KUKA KRL program: MyProgram_120().src

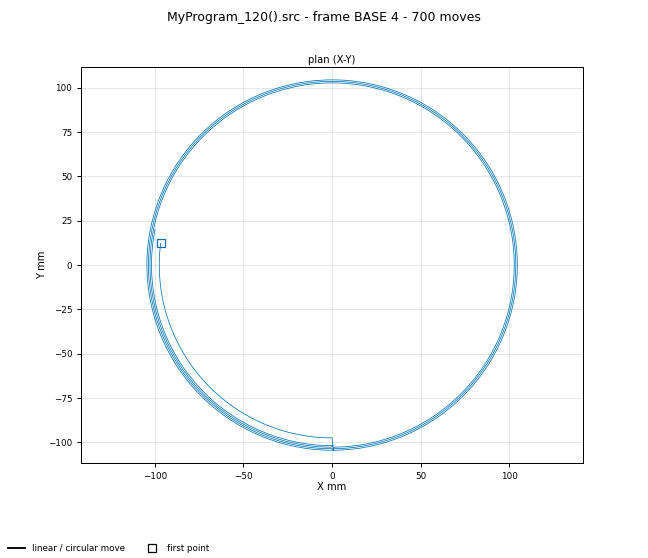
[picture p0: tool path of MyProgram_120().src in frame BASE 4, 700 of 700 moves have a stored position in this frame; points joined in program order, loops and branches not executed]
&ACCESS RVP
&REL 1
&PARAM TEMPLATE = C:\KRC\Roboter\Template\vorgabe
&PARAM EDITMASK = *
DEF MyProgram_120()
; ---- Setting reference (Base) ----
$BASE = BASE_DATA[4]

; --------------------------
; ---- Setting tool (TCP) ----
$TOOL = TOOL_DATA[3]
; --------------------------

$VEL.CP = VEL_APROX_PRINT
Startdeposition()
$VEL.CP = VEL_PRINT
LIN {X -96.7229,Y 12.2113,Z 101,A 168.4745,B 24.9259,C -1.9878,E1 24.8409,E2 276.8389} C_DIS
LIN {X -97.0219,Y 9.5617,Z 101,A 170.028,B 24.9263,C -1.9823,E1 24.8405,E2 275.2892} C_DIS
LIN {X -97.2007,Y 7.5113,Z 101,A 171.291,B 24.9265,C -1.9802,E1 24.8402,E2 274.0237} C_DIS
LIN {X -97.3722,Y 4.8262,Z 101,A 172.8402,B 24.9269,C -1.974,E1 24.8399,E2 272.4798} C_DIS
LIN {X -97.4611,Y 2.4408,Z 101,A 174.2525,B 24.9272,C -1.9698,E1 24.8399,E2 271.0691} C_DIS
LIN {X -97.4919,Y 0.0083,Z 101,A 175.6921,B 24.9276,C -1.9656,E1 24.8398,E2 269.631} C_DIS
LIN {X -97.4637,Y -2.3325,Z 101,A 177.0782,B 24.9279,C -1.9615,E1 24.8398,E2 268.2463} C_DIS
LIN {X -97.3763,Y -4.7434,Z 101,A 178.5071,B 24.9282,C -1.9573,E1 24.84,E2 266.8188} C_DIS
LIN {X -97.231,Y -7.125,Z 101,A 179.9181,B 24.9285,C -1.9531,E1 24.8403,E2 265.4093} C_DIS
LIN {X -97.0288,Y -9.488,Z 101,A -178.679,B 24.9288,C -1.949,E1 24.8407,E2 264.0078} C_DIS
LIN {X -96.7605,Y -11.9197,Z 101,A -177.2313,B 24.9291,C -1.9447,E1 24.8411,E2 262.5616} C_DIS
LIN {X -96.4472,Y -14.2312,Z 101,A -175.8498,B 24.9294,C -1.9408,E1 24.8417,E2 261.1814} C_DIS
LIN {X -96.0565,Y -16.6684,Z 101,A -174.3908,B 24.9297,C -1.9365,E1 24.8423,E2 259.7239} C_DIS
LIN {X -95.6192,Y -19.017,Z 101,A -172.9768,B 24.93,C -1.9324,E1 24.8431,E2 258.3112} C_DIS
LIN {X -95.1138,Y -21.401,Z 101,A -171.3294,B 24.9298,C -1.9351,E1 24.8441,E2 256.6478} C_DIS
LIN {X -94.2834,Y -24.8046,Z 101,A -169.4616,B 24.9307,C -1.9225,E1 24.8453,E2 254.7992} C_DIS
LIN {X -93.6343,Y -27.1534,Z 101,A -168.0199,B 24.931,C -1.9184,E1 24.8464,E2 253.3587} C_DIS
LIN {X -92.6398,Y -30.37,Z 101,A -166.0424,B 24.9314,C -1.9125,E1 24.8481,E2 251.3841} C_DIS
LIN {X -91.9528,Y -32.3885,Z 101,A -164.6967,B 24.9314,C -1.9118,E1 24.8493,E2 250.0322} C_DIS
LIN {X -90.9778,Y -35.038,Z 101,A -163.097,B 24.932,C -1.905,E1 24.8509,E2 248.4399} C_DIS
LIN {X -90.0939,Y -37.2519,Z 101,A -161.6859,B 24.9322,C -1.9012,E1 24.8524,E2 247.0298} C_DIS
LIN {X -89.1565,Y -39.4427,Z 101,A -160.2806,B 24.9325,C -1.8974,E1 24.854,E2 245.626} C_DIS
LIN {X -88.1312,Y -41.6842,Z 101,A -158.8206,B 24.9328,C -1.8937,E1 24.8557,E2 244.1668} C_DIS
LIN {X -87.104,Y -43.7895,Z 101,A -157.4349,B 24.933,C -1.8902,E1 24.8574,E2 242.7821} C_DIS
LIN {X -86.005,Y -45.9104,Z 101,A -155.8779,B 24.933,C -1.8914,E1 24.8594,E2 241.2139} C_DIS
LIN {X -84.4429,Y -48.7212,Z 101,A -154.0565,B 24.9335,C -1.8841,E1 24.8619,E2 239.4005} C_DIS
LIN {X -82.9985,Y -51.1462,Z 101,A -152.4547,B 24.9339,C -1.8777,E1 24.8642,E2 237.8055} C_DIS
LIN {X -81.8862,Y -52.9061,Z 101,A -151.1887,B 24.934,C -1.876,E1 24.8662,E2 236.5372} C_DIS
LIN {X -79.7344,Y -56.0986,Z 101,A -148.9459,B 24.9345,C -1.8696,E1 24.8697,E2 234.2985} C_DIS
LIN {X -78.3085,Y -58.0728,Z 101,A -147.5081,B 24.9347,C -1.8663,E1 24.8721,E2 232.8617} C_DIS
LIN {X -76.7454,Y -60.1219,Z 101,A -145.8271,B 24.9346,C -1.8683,E1 24.875,E2 231.1679} C_DIS
LIN {X -74.5735,Y -62.7968,Z 101,A -143.7539,B 24.9348,C -1.8652,E1 24.8787,E2 229.0926} C_DIS
LIN {X -72.2811,Y -65.4221,Z 101,A -141.6893,B 24.9351,C -1.8611,E1 24.8825,E2 227.0285} C_DIS
LIN {X -70.1933,Y -67.6552,Z 101,A -139.9774,B 24.9355,C -1.8543,E1 24.8858,E2 225.3253} C_DIS
LIN {X -67.6749,Y -70.1743,Z 101,A -137.8668,B 24.9358,C -1.8505,E1 24.89,E2 223.2149} C_DIS
LIN {X -65.0221,Y -72.6391,Z 101,A -135.7428,B 24.9361,C -1.8461,E1 24.8943,E2 221.0927} C_DIS
LIN {X -62.3326,Y -74.9598,Z 101,A -133.6387,B 24.9364,C -1.8427,E1 24.8988,E2 218.9887} C_DIS
LIN {X -59.5972,Y -77.1525,Z 101,A -131.585,B 24.9366,C -1.8387,E1 24.9033,E2 216.9369} C_DIS
LIN {X -57.1512,Y -78.9834,Z 101,A -129.8771,B 24.9371,C -1.8326,E1 24.9071,E2 215.2376} C_DIS
LIN {X -55.1551,Y -80.3903,Z 101,A -128.4366,B 24.9372,C -1.8304,E1 24.9105,E2 213.7974} C_DIS
LIN {X -53.1374,Y -81.7378,Z 101,A -126.7931,B 24.9368,C -1.8357,E1 24.9143,E2 212.1358} C_DIS
LIN {X -50.1638,Y -83.5955,Z 101,A -124.9406,B 24.9375,C -1.8254,E1 24.9187,E2 210.3021} C_DIS
LIN {X -48.0882,Y -84.8066,Z 101,A -123.5216,B 24.9377,C -1.8236,E1 24.9221,E2 208.8832} C_DIS
LIN {X -45.9565,Y -85.9807,Z 101,A -122.0876,B 24.9377,C -1.8218,E1 24.9257,E2 207.4493} C_DIS
LIN {X -42.7678,Y -87.6104,Z 101,A -119.9768,B 24.938,C -1.8194,E1 24.9309,E2 205.3386} C_DIS
LIN {X -40.652,Y -88.6117,Z 101,A -118.5977,B 24.938,C -1.818,E1 24.9344,E2 203.9595} C_DIS
LIN {X -38.4283,Y -89.5987,Z 101,A -117.1645,B 24.9381,C -1.8166,E1 24.9381,E2 202.5263} C_DIS
LIN {X -36.5181,Y -90.3926,Z 101,A -115.9075,B 24.9381,C -1.8168,E1 24.9413,E2 201.2659} C_DIS
LIN {X -34.0204,Y -91.3632,Z 101,A -114.3685,B 24.9383,C -1.8141,E1 24.9453,E2 199.7302} C_DIS
LIN {X -31.8745,Y -92.1332,Z 101,A -113.0168,B 24.9383,C -1.8134,E1 24.9489,E2 198.3775} C_DIS
LIN {X -29.4455,Y -92.9389,Z 101,A -111.5188,B 24.9385,C -1.812,E1 24.9529,E2 196.8801} C_DIS
LIN {X -27.1599,Y -93.6323,Z 101,A -110.1131,B 24.9385,C -1.8111,E1 24.9567,E2 195.4743} C_DIS
LIN {X -24.8583,Y -94.2695,Z 101,A -108.7074,B 24.9385,C -1.8103,E1 24.9604,E2 194.0682} C_DIS
LIN {X -22.864,Y -94.7714,Z 101,A -107.4594,B 24.9385,C -1.811,E1 24.9638,E2 192.8167} C_DIS
LIN {X -20.1943,Y -95.3775,Z 101,A -105.8867,B 24.9387,C -1.809,E1 24.9681,E2 191.2469} C_DIS
LIN {X -17.8998,Y -95.8343,Z 101,A -104.5109,B 24.9387,C -1.8085,E1 24.9719,E2 189.8707} C_DIS
LIN {X -15.5499,Y -96.2435,Z 101,A -103.1064,B 24.9387,C -1.8082,E1 24.9758,E2 188.4658} C_DIS
LIN {X -13.179,Y -96.5967,Z 101,A -101.6986,B 24.9387,C -1.8078,E1 24.9797,E2 187.0577} C_DIS
LIN {X -10.8195,Y -96.8893,Z 101,A -100.0943,B 24.9382,C -1.8151,E1 24.9842,E2 185.4349} C_DIS
LIN {X -7.2888,Y -97.2185,Z 101,A -98.2167,B 24.9388,C -1.8075,E1 24.9893,E2 183.5745} C_DIS
LIN {X -5.0349,Y -97.3606,Z 101,A -96.9033,B 24.9388,C -1.8071,E1 24.993,E2 182.2616} C_DIS
LIN {X -2.4398,Y -97.4611,Z 101,A -95.3423,B 24.9387,C -1.8085,E1 24.9974,E2 180.6971} C_DIS
LIN {X -0.0255,Y -97.4918,Z 101,A -93.9449,B 24.9387,C -1.8081,E1 25.0013,E2 179.3007} C_DIS
LIN {X -0.0255,Y -97.4918,Z 101,A -93.9449,B 24.9387,C -1.8081,E1 25.0013,E2 179.3007} C_DIS
Enddeposition()
LIN {X 0.7251,Y -104.456,Z 102,A -93.6482,B 24.9465,C -1.6893,E1 25.0013,E2 179.2858} C_DIS
Startdeposition()
$VEL.CP = VEL_PRINT
LIN {X 2.706,Y -104.4247,Z 102,A -92.2701,B 24.9458,C -1.7011,E1 25.0052,E2 177.8798} C_DIS
LIN {X 5.2679,Y -104.3268,Z 102,A -90.7936,B 24.9456,C -1.7044,E1 25.0094,E2 176.3959} C_DIS
LIN {X 7.8267,Y -104.1661,Z 102,A -89.46,B 24.9457,C -1.7022,E1 25.0131,E2 175.0683} C_DIS
LIN {X 10.7597,Y -103.903,Z 102,A -87.9361,B 24.9459,C -1.6994,E1 25.0173,E2 173.5518} C_DIS
LIN {X 12.7871,Y -103.6749,Z 102,A -86.5933,B 24.9453,C -1.709,E1 25.0211,E2 172.1872} C_DIS
LIN {X 15.4684,Y -103.3081,Z 102,A -85.045,B 24.945,C -1.7126,E1 25.0254,E2 170.6318} C_DIS
LIN {X 20.3792,Y -102.4533,Z 102,A -82.4457,B 24.9452,C -1.7094,E1 25.0325,E2 168.0431} C_DIS
LIN {X 23.0263,Y -101.8902,Z 102,A -81.0356,B 24.9453,C -1.7077,E1 25.0363,E2 166.6387} C_DIS
LIN {X 25.5972,Y -101.2746,Z 102,A -79.5528,B 24.9452,C -1.7105,E1 25.0403,E2 165.1514} C_DIS
LIN {X 27.8609,Y -100.6765,Z 102,A -78.1735,B 24.9448,C -1.7157,E1 25.0441,E2 163.762} C_DIS
LIN {X 30.4594,Y -99.9202,Z 102,A -76.827,B 24.9451,C -1.7118,E1 25.0477,E2 162.4271} C_DIS
LIN {X 32.9024,Y -99.1426,Z 102,A -75.229,B 24.9445,C -1.7214,E1 25.052,E2 160.8095} C_DIS
LIN {X 36.396,Y -97.9149,Z 102,A -73.2633,B 24.9445,C -1.7214,E1 25.0571,E2 158.8479} C_DIS
LIN {X 38.788,Y -96.9922,Z 102,A -71.8613,B 24.9444,C -1.7231,E1 25.0607,E2 157.4449} C_DIS
LIN {X 41.1566,Y -96.0111,Z 102,A -70.5237,B 24.9444,C -1.7224,E1 25.0642,E2 156.1121} C_DIS
LIN {X 43.5004,Y -94.9721,Z 102,A -69.058,B 24.9441,C -1.727,E1 25.0679,E2 154.6392} C_DIS
LIN {X 45.9458,Y -93.8127,Z 102,A -67.6428,B 24.9441,C -1.7266,E1 25.0715,E2 153.2288} C_DIS
LIN {X 48.2342,Y -92.6569,Z 102,A -66.3132,B 24.9441,C -1.7258,E1 25.0748,E2 151.9047} C_DIS
LIN {X 50.3692,Y -91.5147,Z 102,A -64.8544,B 24.9437,C -1.7335,E1 25.0784,E2 150.4319} C_DIS
LIN {X 52.5999,Y -90.251,Z 102,A -63.32,B 24.9432,C -1.7413,E1 25.0821,E2 148.8835} C_DIS
LIN {X 54.9198,Y -88.8575,Z 102,A -62.0393,B 24.9435,C -1.7357,E1 25.0851,E2 147.6202} C_DIS
LIN {X 57.0839,Y -87.4829,Z 102,A -60.639,B 24.9434,C -1.7382,E1 25.0884,E2 146.2186} C_DIS
LIN {X 59.3797,Y -85.9402,Z 102,A -59.3008,B 24.9437,C -1.7338,E1 25.0915,E2 144.8952} C_DIS
LIN {X 61.1927,Y -84.6608,Z 102,A -57.9169,B 24.943,C -1.7432,E1 25.0947,E2 143.4939} C_DIS
LIN {X 63.252,Y -83.1335,Z 102,A -56.3188,B 24.9423,C -1.7542,E1 25.0983,E2 141.8756} C_DIS
LIN {X 65.8495,Y -81.0891,Z 102,A -54.6326,B 24.9424,C -1.7529,E1 25.1019,E2 140.1988} C_DIS
LIN {X 68.2308,Y -79.0984,Z 102,A -53.0182,B 24.9424,C -1.7531,E1 25.1053,E2 138.5903} C_DIS
LIN {X 70.2564,Y -77.3038,Z 102,A -51.6126,B 24.9424,C -1.7533,E1 25.1083,E2 137.1899} C_DIS
LIN {X 72.1324,Y -75.5563,Z 102,A -50.1267,B 24.9419,C -1.7599,E1 25.1113,E2 135.6943} C_DIS
LIN {X 73.9649,Y -73.7633,Z 102,A -48.8148,B 24.9419,C -1.7594,E1 25.1139,E2 134.3892} C_DIS
LIN {X 75.7528,Y -71.9259,Z 102,A -47.416,B 24.9418,C -1.7626,E1 25.1166,E2 132.989} C_DIS
LIN {X 77.4952,Y -70.0452,Z 102,A -45.9461,B 24.9414,C -1.7688,E1 25.1194,E2 131.5107} C_DIS
LIN {X 79.0984,Y -68.2308,Z 102,A -44.6253,B 24.9412,C -1.772,E1 25.1218,E2 130.1886} C_DIS
LIN {X 80.749,Y -66.269,Z 102,A -43.1634,B 24.9407,C -1.778,E1 25.1244,E2 128.7191} C_DIS
LIN {X 82.4381,Y -64.1545,Z 102,A -41.7513,B 24.9407,C -1.7789,E1 25.1269,E2 127.3114} C_DIS
LIN {X 83.9877,Y -62.112,Z 102,A -40.3534,B 24.9405,C -1.7824,E1 25.1292,E2 125.912} C_DIS
LIN {X 85.4867,Y -60.0322,Z 102,A -39.0265,B 24.9405,C -1.783,E1 25.1313,E2 124.5903} C_DIS
LIN {X 86.8557,Y -58.0351,Z 102,A -37.5514,B 24.9398,C -1.7929,E1 25.1337,E2 123.0991} C_DIS
LIN {X 88.3541,Y -55.7256,Z 102,A -36.2293,B 24.94,C -1.7892,E1 25.1356,E2 121.7922} C_DIS
LIN {X 89.6713,Y -53.5807,Z 102,A -34.8339,B 24.9397,C -1.7938,E1 25.1377,E2 120.3931} C_DIS
LIN {X 90.9592,Y -51.3639,Z 102,A -33.3656,B 24.9392,C -1.8006,E1 25.1397,E2 118.9165} C_DIS
LIN {X 92.1259,Y -49.2423,Z 102,A -32.0454,B 24.939,C -1.8041,E1 25.1415,E2 117.5948} C_DIS
LIN {X 93.3066,Y -46.9666,Z 102,A -30.5705,B 24.9385,C -1.8113,E1 25.1434,E2 116.1109} C_DIS
LIN {X 94.4913,Y -44.5334,Z 102,A -29.1738,B 24.9385,C -1.812,E1 25.145,E2 114.72} C_DIS
LIN {X 95.5558,Y -42.2011,Z 102,A -27.8476,B 24.9384,C -1.8129,E1 25.1466,E2 113.3989} C_DIS
LIN {X 96.5626,Y -39.8433,Z 102,A -26.4507,B 24.9381,C -1.8168,E1 25.1481,E2 112.0005} C_DIS
LIN {X 97.5114,Y -37.4615,Z 102,A -24.9829,B 24.9377,C -1.8238,E1 25.1496,E2 110.5244} C_DIS
LIN {X 98.3542,Y -35.1917,Z 102,A -23.5661,B 24.9371,C -1.8317,E1 25.1509,E2 109.0969} C_DIS
LIN {X 99.2321,Y -32.6317,Z 102,A -22.2603,B 24.9373,C -1.8287,E1 25.1521,E2 107.8054} C_DIS
LIN {X 100.003,Y -30.1866,Z 102,A -20.7927,B 24.9368,C -1.8358,E1 25.1533,E2 106.3296} C_DIS
LIN {X 100.6765,Y -27.8609,Z 102,A -19.2824,B 24.936,C -1.8477,E1 25.1544,E2 104.7996} C_DIS
LIN {X 101.3637,Y -25.2434,Z 102,A -18.0701,B 24.9365,C -1.8409,E1 25.1553,E2 103.6106} C_DIS
LIN {X 101.9527,Y -22.7482,Z 102,A -16.4523,B 24.9355,C -1.8544,E1 25.1563,E2 101.9702} C_DIS
LIN {X 102.7209,Y -18.9802,Z 102,A -14.5079,B 24.9355,C -1.8541,E1 25.1573,E2 100.0379} C_DIS
LIN {X 103.134,Y -16.5944,Z 102,A -13.1889,B 24.9353,C -1.858,E1 25.1579,E2 98.7175} C_DIS
LIN {X 103.5285,Y -13.917,Z 102,A -11.7862,B 24.9352,C -1.8593,E1 25.1585,E2 97.3198} C_DIS
LIN {X 103.824,Y -11.5139,Z 102,A -10.3321,B 24.9345,C -1.869,E1 25.1589,E2 95.8516} C_DIS
LIN {X 104.0753,Y -8.9624,Z 102,A -8.9997,B 24.9345,C -1.8704,E1 25.1593,E2 94.5238} C_DIS
LIN {X 104.2639,Y -6.4056,Z 102,A -7.5393,B 24.9339,C -1.8773,E1 25.1596,E2 93.0558} C_DIS
LIN {X 104.3897,Y -3.8449,Z 102,A -6.1429,B 24.9336,C -1.8814,E1 25.1597,E2 91.658} C_DIS
LIN {X 104.4526,Y -1.2819,Z 102,A -4.7464,B 24.9334,C -1.8855,E1 25.1597,E2 90.2601} C_DIS
LIN {X 104.4526,Y 1.2819,Z 102,A -3.35,B 24.9331,C -1.8896,E1 25.1597,E2 88.8622} C_DIS
LIN {X 104.3897,Y 3.8449,Z 102,A -2.0172,B 24.933,C -1.891,E1 25.1597,E2 87.5341} C_DIS
LIN {X 104.2543,Y 6.5478,Z 102,A -0.5432,B 24.9327,C -1.8954,E1 25.1594,E2 86.0586} C_DIS
LIN {X 104.0622,Y 9.1044,Z 102,A 0.782,B 24.9326,C -1.8964,E1 25.1591,E2 84.7388} C_DIS
LIN {X 103.8074,Y 11.6554,Z 102,A 2.1787,B 24.9323,C -1.9005,E1 25.1587,E2 83.3407} C_DIS
LIN {X 103.4901,Y 14.1995,Z 102,A 3.7088,B 24.9316,C -1.9103,E1 25.1581,E2 81.7967} C_DIS
LIN {X 103.134,Y 16.5944,Z 102,A 5.0569,B 24.9312,C -1.9153,E1 25.1576,E2 80.4446} C_DIS
LIN {X 102.6687,Y 19.2604,Z 102,A 6.3687,B 24.9314,C -1.9126,E1 25.1569,E2 79.1468} C_DIS
LIN {X 102.1651,Y 21.7742,Z 102,A 7.9938,B 24.9304,C -1.9263,E1 25.156,E2 77.4989} C_DIS
LIN {X 101.2945,Y 25.5199,Z 102,A 9.9321,B 24.9304,C -1.9256,E1 25.1547,E2 75.5735} C_DIS
LIN {X 100.6765,Y 27.8609,Z 102,A 11.2512,B 24.9302,C -1.9292,E1 25.1537,E2 74.2534} C_DIS
LIN {X 99.8974,Y 30.5331,Z 102,A 12.7342,B 24.93,C -1.9321,E1 25.1526,E2 72.7722} C_DIS
LIN {X 99.1882,Y 32.7673,Z 102,A 14.1096,B 24.9295,C -1.9397,E1 25.1514,E2 71.3866} C_DIS
LIN {X 98.3542,Y 35.1917,Z 102,A 15.5068,B 24.9292,C -1.9435,E1 25.1501,E2 69.9883} C_DIS
LIN {X 97.4609,Y 37.5948,Z 102,A 16.9042,B 24.9289,C -1.9473,E1 25.1487,E2 68.5898} C_DIS
LIN {X 96.4536,Y 40.1066,Z 102,A 18.3337,B 24.9288,C -1.9493,E1 25.1472,E2 67.1633} C_DIS
LIN {X 95.4402,Y 42.4616,Z 102,A 19.7128,B 24.9285,C -1.9522,E1 25.1456,E2 65.785} C_DIS
LIN {X 94.3694,Y 44.7911,Z 102,A 21.0392,B 24.9285,C -1.9528,E1 25.1441,E2 64.4642} C_DIS
LIN {X 93.2418,Y 47.0935,Z 102,A 22.5323,B 24.9279,C -1.9604,E1 25.1422,E2 62.9612} C_DIS
LIN {X 92.058,Y 49.3676,Z 102,A 23.9058,B 24.9278,C -1.9629,E1 25.1404,E2 61.589} C_DIS
LIN {X 90.8897,Y 51.4884,Z 102,A 25.2263,B 24.9275,C -1.9662,E1 25.1386,E2 60.2676} C_DIS
LIN {X 89.5987,Y 53.7034,Z 102,A 26.6881,B 24.9271,C -1.9723,E1 25.1365,E2 58.799} C_DIS
LIN {X 88.0916,Y 56.1388,Z 102,A 28.0368,B 24.9274,C -1.9671,E1 25.1345,E2 57.4692} C_DIS
LIN {X 86.7357,Y 58.2123,Z 102,A 29.5065,B 24.9268,C -1.9752,E1 25.1323,E2 55.9877} C_DIS
LIN {X 85.4053,Y 60.1492,Z 102,A 30.8904,B 24.9263,C -1.9825,E1 25.13,E2 54.5935} C_DIS
LIN {X 83.8179,Y 62.341,Z 102,A 32.225,B 24.9265,C -1.9799,E1 25.1278,E2 53.2714} C_DIS
LIN {X 82.2305,Y 64.42,Z 102,A 33.6263,B 24.9263,C -1.982,E1 25.1255,E2 51.8717} C_DIS
LIN {X 80.7491,Y 66.269,Z 102,A 35.0163,B 24.9258,C -1.9888,E1 25.123,E2 50.4721} C_DIS
LIN {X 78.8179,Y 68.5519,Z 102,A 36.5266,B 24.9259,C -1.9873,E1 25.1203,E2 48.9723} C_DIS
LIN {X 77.3038,Y 70.2564,Z 102,A 37.8212,B 24.9256,C -1.992,E1 25.1179,E2 47.6724} C_DIS
LIN {X 75.6552,Y 72.0297,Z 102,A 39.391,B 24.9246,C -2.0049,E1 25.1148,E2 46.079} C_DIS
LIN {X 73.3658,Y 74.3575,Z 102,A 41.0872,B 24.9246,C -2.0049,E1 25.1115,E2 44.39} C_DIS
LIN {X 70.9909,Y 76.6298,Z 102,A 42.7915,B 24.9246,C -2.0045,E1 25.108,E2 42.6936} C_DIS
LIN {X 69.1963,Y 78.2552,Z 102,A 44.1141,B 24.9245,C -2.0069,E1 25.1053,E2 41.3705} C_DIS
LIN {X 67.255,Y 79.9297,Z 102,A 45.5144,B 24.9243,C -2.0094,E1 25.1023,E2 39.9698} C_DIS
LIN {X 65.2731,Y 81.5562,Z 102,A 46.9789,B 24.9239,C -2.0144,E1 25.0991,E2 38.499} C_DIS
LIN {X 63.252,Y 83.1335,Z 102,A 48.38,B 24.9237,C -2.0167,E1 25.096,E2 37.0975} C_DIS
LIN {X 61.0597,Y 84.7556,Z 102,A 49.7244,B 24.924,C -2.0132,E1 25.093,E2 35.7663} C_DIS
LIN {X 59.0966,Y 86.137,Z 102,A 51.182,B 24.9234,C -2.0211,E1 25.0896,E2 34.2949} C_DIS
LIN {X 56.9649,Y 87.5614,Z 102,A 52.5833,B 24.9232,C -2.0232,E1 25.0863,E2 32.8934} C_DIS
LIN {X 54.6771,Y 89.007,Z 102,A 53.9987,B 24.9232,C -2.0226,E1 25.083,E2 31.4837} C_DIS
LIN {X 51.4884,Y 90.8897,Z 102,A 56.0234,B 24.9231,C -2.0253,E1 25.0781,E2 29.4588} C_DIS
LIN {X 49.1162,Y 92.1923,Z 102,A 57.4323,B 24.9231,C -2.0243,E1 25.0747,E2 28.0564} C_DIS
LIN {X 46.8389,Y 93.3699,Z 102,A 59.0377,B 24.9224,C -2.0341,E1 25.0706,E2 26.432} C_DIS
LIN {X 43.5004,Y 94.9721,Z 102,A 60.9319,B 24.9226,C -2.031,E1 25.0659,E2 24.5501} C_DIS
LIN {X 41.1566,Y 96.0111,Z 102,A 62.3989,B 24.9223,C -2.035,E1 25.0621,E2 23.0772} C_DIS
LIN {X 38.788,Y 96.9922,Z 102,A 63.7377,B 24.9224,C -2.0338,E1 25.0586,E2 21.7444} C_DIS
LIN {X 36.2621,Y 97.9637,Z 102,A 65.1474,B 24.9226,C -2.0322,E1 25.055,E2 20.3413} C_DIS
LIN {X 33.9821,Y 98.7786,Z 102,A 66.6088,B 24.9221,C -2.0387,E1 25.0511,E2 18.8676} C_DIS
LIN {X 31.5477,Y 99.5828,Z 102,A 67.9485,B 24.9221,C -2.0372,E1 25.0476,E2 17.534} C_DIS
LIN {X 28.9572,Y 100.3659,Z 102,A 69.3588,B 24.9223,C -2.0354,E1 25.0438,E2 16.1305} C_DIS
LIN {X 26.6234,Y 101.0108,Z 102,A 70.8209,B 24.9218,C -2.0415,E1 25.0398,E2 14.6562} C_DIS
LIN {X 24.1364,Y 101.6338,Z 102,A 72.2253,B 24.9218,C -2.0422,E1 25.036,E2 13.252} C_DIS
LIN {X 21.4953,Y 102.2242,Z 102,A 73.5723,B 24.9221,C -2.0376,E1 25.0324,E2 11.9179} C_DIS
LIN {X 18.9802,Y 102.7209,Z 102,A 75.0489,B 24.9219,C -2.0409,E1 25.0283,E2 10.4351} C_DIS
LIN {X 16.4535,Y 103.1558,Z 102,A 76.3827,B 24.9221,C -2.0385,E1 25.0246,E2 9.1082} C_DIS
LIN {X 13.7479,Y 103.5504,Z 102,A 77.7958,B 24.9223,C -2.0356,E1 25.0208,E2 7.7035} C_DIS
LIN {X 11.5139,Y 103.824,Z 102,A 79.2518,B 24.9216,C -2.0444,E1 25.0167,E2 6.2276} C_DIS
LIN {X 8.9624,Y 104.0753,Z 102,A 80.5931,B 24.9218,C -2.042,E1 25.013,E2 4.8927} C_DIS
LIN {X 6.4056,Y 104.2639,Z 102,A 82.0638,B 24.9216,C -2.0445,E1 25.0088,E2 3.4166} C_DIS
LIN {X 3.8449,Y 104.3897,Z 102,A 83.4702,B 24.9216,C -2.0445,E1 25.0049,E2 2.0108} C_DIS
LIN {X 1.0654,Y 104.454,Z 102,A 84.8985,B 24.9219,C -2.0405,E1 25.001,E2 0.5921} C_DIS
LIN {X -1.2819,Y 104.4526,Z 102,A 86.2838,B 24.9217,C -2.044,E1 24.9971,E2 -0.8015} C_DIS
LIN {X -3.8449,Y 104.3897,Z 102,A 87.6912,B 24.9217,C -2.0436,E1 24.9931,E2 -2.2081} C_DIS
LIN {X -6.5478,Y 104.2543,Z 102,A 89.1122,B 24.9219,C -2.0406,E1 24.9892,E2 -3.6225} C_DIS
LIN {X -8.9624,Y 104.0753,Z 102,A 90.506,B 24.9218,C -2.0425,E1 24.9853,E2 -5.0215} C_DIS
LIN {X -11.6554,Y 103.8074,Z 102,A 91.8558,B 24.9222,C -2.0366,E1 24.9816,E2 -6.3581} C_DIS
LIN {X -14.1995,Y 103.4901,Z 102,A 93.3358,B 24.9221,C -2.0386,E1 24.9775,E2 -7.8438} C_DIS
LIN {X -16.9865,Y 103.0684,Z 102,A 94.6843,B 24.9227,C -2.03,E1 24.9738,E2 -9.1731} C_DIS
LIN {X -19.2604,Y 102.6687,Z 102,A 96.1463,B 24.9222,C -2.0364,E1 24.9697,E2 -10.6519} C_DIS
LIN {X -21.635,Y 102.1955,Z 102,A 97.5477,B 24.9222,C -2.0381,E1 24.9659,E2 -12.0589} C_DIS
LIN {X -24.1364,Y 101.6338,Z 102,A 98.9568,B 24.9222,C -2.0369,E1 24.9621,E2 -13.467} C_DIS
LIN {X -26.761,Y 100.9737,Z 102,A 100.4367,B 24.9223,C -2.0353,E1 24.9581,E2 -14.9452} C_DIS
LIN {X -29.0943,Y 100.327,Z 102,A 101.776,B 24.9224,C -2.0342,E1 24.9545,E2 -16.2842} C_DIS
LIN {X -31.5477,Y 99.5828,Z 102,A 103.1854,B 24.9225,C -2.0328,E1 24.9507,E2 -17.6925} C_DIS
LIN {X -34.1166,Y 98.7314,Z 102,A 104.5373,B 24.923,C -2.026,E1 24.9472,E2 -19.0309} C_DIS
LIN {X -36.5293,Y 97.8644,Z 102,A 106.0194,B 24.923,C -2.027,E1 24.9433,E2 -20.5185} C_DIS
LIN {X -38.788,Y 96.9922,Z 102,A 107.4161,B 24.9229,C -2.0278,E1 24.9396,E2 -21.9199} C_DIS
LIN {X -41.1566,Y 96.0111,Z 102,A 108.7621,B 24.9232,C -2.0235,E1 24.9362,E2 -23.2589} C_DIS
LIN {X -43.5004,Y 94.9721,Z 102,A 110.2377,B 24.9232,C -2.024,E1 24.9324,E2 -24.7392} C_DIS
LIN {X -45.9458,Y 93.8127,Z 102,A 111.6928,B 24.9234,C -2.0205,E1 24.9288,E2 -26.1899} C_DIS
LIN {X -48.2342,Y 92.6569,Z 102,A 113.0736,B 24.9237,C -2.0173,E1 24.9254,E2 -27.5668} C_DIS
LIN {X -50.3692,Y 91.5147,Z 102,A 114.4071,B 24.9239,C -2.0152,E1 24.9221,E2 -28.8991} C_DIS
LIN {X -52.8041,Y 90.1303,Z 102,A 115.9072,B 24.9242,C -2.0111,E1 24.9185,E2 -30.3939} C_DIS
LIN {X -54.9198,Y 88.8575,Z 102,A 117.3091,B 24.9242,C -2.0104,E1 24.9151,E2 -31.7984} C_DIS
LIN {X -57.0888,Y 87.4797,Z 102,A 118.7217,B 24.9244,C -2.0078,E1 24.9118,E2 -33.2094} C_DIS
LIN {X -59.0966,Y 86.137,Z 102,A 120.1128,B 24.9244,C -2.0076,E1 24.9086,E2 -34.6048} C_DIS
LIN {X -61.1927,Y 84.6608,Z 102,A 121.5321,B 24.9246,C -2.0052,E1 24.9054,E2 -36.0233} C_DIS
LIN {X -63.252,Y 83.1335,Z 102,A 122.8798,B 24.925,C -2.0002,E1 24.9024,E2 -37.3638} C_DIS
LIN {X -65.3839,Y 81.4665,Z 102,A 124.3713,B 24.9252,C -1.9972,E1 24.8991,E2 -38.8537} C_DIS
LIN {X -67.3634,Y 79.8373,Z 102,A 125.7844,B 24.9254,C -1.9944,E1 24.8961,E2 -40.2654} C_DIS
LIN {X -69.1963,Y 78.2552,Z 102,A 127.1839,B 24.9254,C -1.9939,E1 24.8931,E2 -41.6695} C_DIS
LIN {X -71.0959,Y 76.5334,Z 102,A 128.5973,B 24.9257,C -1.9909,E1 24.8902,E2 -43.0814} C_DIS
LIN {X -72.9527,Y 74.7656,Z 102,A 130.011,B 24.9259,C -1.9878,E1 24.8874,E2 -44.4937} C_DIS
LIN {X -74.8645,Y 72.8501,Z 102,A 131.4381,B 24.9263,C -1.9822,E1 24.8846,E2 -45.9133} C_DIS
LIN {X -76.5334,Y 71.0959,Z 102,A 132.7736,B 24.9266,C -1.9791,E1 24.8821,E2 -47.2474} C_DIS
LIN {X -78.2552,Y 69.1963,Z 102,A 134.2525,B 24.9266,C -1.9782,E1 24.8793,E2 -48.7306} C_DIS
LIN {X -80.0208,Y 67.1453,Z 102,A 135.6803,B 24.9271,C -1.9723,E1 24.8767,E2 -50.151} C_DIS
LIN {X -81.6446,Y 65.1613,Z 102,A 137.0948,B 24.9273,C -1.9689,E1 24.8743,E2 -51.564} C_DIS
LIN {X -83.2191,Y 63.138,Z 102,A 138.4372,B 24.9278,C -1.9629,E1 24.872,E2 -52.8983} C_DIS
LIN {X -84.7435,Y 61.0767,Z 102,A 139.8519,B 24.928,C -1.9593,E1 24.8697,E2 -54.3115} C_DIS
LIN {X -86.4165,Y 58.6838,Z 102,A 141.3827,B 24.9285,C -1.9524,E1 24.8673,E2 -55.8333} C_DIS
LIN {X -87.6384,Y 56.845,Z 102,A 142.6814,B 24.9285,C -1.9521,E1 24.8652,E2 -57.1378} C_DIS
LIN {X -88.9592,Y 54.7558,Z 102,A 144.1595,B 24.9285,C -1.9526,E1 24.863,E2 -58.6248} C_DIS
LIN {X -90.251,Y 52.5999,Z 102,A 145.57,B 24.9287,C -1.9498,E1 24.8611,E2 -60.0358} C_DIS
LIN {X -91.5827,Y 50.2439,Z 102,A 146.9989,B 24.9292,C -1.9435,E1 24.8591,E2 -61.4572} C_DIS
LIN {X -92.7233,Y 48.1081,Z 102,A 148.4004,B 24.9292,C -1.9422,E1 24.8573,E2 -62.8631} C_DIS
LIN {X -93.876,Y 45.8181,Z 102,A 149.8938,B 24.9294,C -1.9412,E1 24.8554,E2 -64.362} C_DIS
LIN {X -94.9721,Y 43.5004,Z 102,A 151.2312,B 24.9298,C -1.9345,E1 24.8539,E2 -65.6907} C_DIS
LIN {X -96.0664,Y 41.0253,Z 102,A 152.5886,B 24.9305,C -1.9254,E1 24.8524,E2 -67.0341} C_DIS
LIN {X -96.9922,Y 38.788,Z 102,A 154.0625,B 24.9305,C -1.9266,E1 24.8508,E2 -68.5189} C_DIS
LIN {X -97.9637,Y 36.2621,Z 102,A 155.4198,B 24.9311,C -1.9175,E1 24.8495,E2 -69.8621} C_DIS
LIN {X -98.8241,Y 33.847,Z 102,A 156.9078,B 24.9311,C -1.916,E1 24.8481,E2 -71.3551} C_DIS
LIN {X -99.625,Y 31.4116,Z 102,A 158.3237,B 24.9315,C -1.9119,E1 24.8469,E2 -72.7694} C_DIS
LIN {X -100.327,Y 29.0943,Z 102,A 159.6611,B 24.9317,C -1.9081,E1 24.8459,E2 -74.1053} C_DIS
LIN {X -101.1253,Y 26.178,Z 102,A 161.1939,B 24.9324,C -1.8984,E1 24.8448,E2 -75.624} C_DIS
LIN {X -101.6338,Y 24.1364,Z 102,A 162.558,B 24.9322,C -1.9022,E1 24.8439,E2 -77.005} C_DIS
LIN {X -102.2242,Y 21.4953,Z 102,A 164.1409,B 24.9322,C -1.9009,E1 24.8429,E2 -78.5944} C_DIS
LIN {X -102.9461,Y 17.7182,Z 102,A 166.1119,B 24.9331,C -1.8892,E1 24.8419,E2 -80.5491} C_DIS
LIN {X -103.3299,Y 15.3275,Z 102,A 167.5143,B 24.9332,C -1.8876,E1 24.8413,E2 -81.956} C_DIS
LIN {X -103.727,Y 12.3421,Z 102,A 168.9809,B 24.934,C -1.8757,E1 24.8408,E2 -83.403} C_DIS
LIN {X -103.9575,Y 10.2389,Z 102,A 170.282,B 24.934,C -1.8769,E1 24.8405,E2 -84.7148} C_DIS
LIN {X -104.1775,Y 7.6846,Z 102,A 171.7627,B 24.934,C -1.8751,E1 24.8401,E2 -86.1999} C_DIS
LIN {X -104.3408,Y 4.9832,Z 102,A 173.1205,B 24.9347,C -1.8658,E1 24.8399,E2 -87.5437} C_DIS
LIN {X -104.4317,Y 2.4211,Z 102,A 174.5369,B 24.935,C -1.8616,E1 24.8399,E2 -88.9587} C_DIS
LIN {X -104.4596,Y -0.1425,Z 102,A 175.953,B 24.9353,C -1.8574,E1 24.8398,E2 -90.3733} C_DIS
LIN {X -104.4247,Y -2.706,Z 102,A 177.3691,B 24.9356,C -1.8532,E1 24.8398,E2 -91.7881} C_DIS
LIN {X -104.3268,Y -5.2679,Z 102,A 178.8573,B 24.9357,C -1.8516,E1 24.84,E2 -93.2813} C_DIS
LIN {X -104.1661,Y -7.8267,Z 102,A -179.7986,B 24.9362,C -1.8449,E1 24.8403,E2 -94.6175} C_DIS
LIN {X -103.9399,Y -10.4064,Z 102,A -178.3081,B 24.9363,C -1.8429,E1 24.8407,E2 -96.1122} C_DIS
LIN {X -103.6749,Y -12.7871,Z 102,A -176.9082,B 24.9364,C -1.8418,E1 24.8412,E2 -97.5178} C_DIS
LIN {X -103.3081,Y -15.4684,Z 102,A -175.5508,B 24.9371,C -1.8326,E1 24.8417,E2 -98.8612} C_DIS
LIN {X -102.9226,Y -17.8588,Z 102,A -174.0764,B 24.937,C -1.8336,E1 24.8424,E2 -100.3469} C_DIS
LIN {X -102.4533,Y -20.3792,Z 102,A -172.7253,B 24.9374,C -1.8272,E1 24.8431,E2 -101.6909} C_DIS
LIN {X -101.8902,Y -23.0263,Z 102,A -171.3029,B 24.9379,C -1.8204,E1 24.8439,E2 -103.1054} C_DIS
LIN {X -101.2945,Y -25.5199,Z 102,A -169.8152,B 24.9379,C -1.819,E1 24.8449,E2 -104.5984} C_DIS
LIN {X -100.6765,Y -27.8609,Z 102,A -168.3794,B 24.9379,C -1.8188,E1 24.846,E2 -106.042} C_DIS
LIN {X -99.9202,Y -30.4594,Z 102,A -167.0563,B 24.9387,C -1.8085,E1 24.847,E2 -107.3482} C_DIS
LIN {X -99.1426,Y -32.9024,Z 102,A -165.5685,B 24.9387,C -1.8073,E1 24.8483,E2 -108.8416} C_DIS
LIN {X -98.3542,Y -35.1917,Z 102,A -164.2319,B 24.939,C -1.8036,E1 24.8495,E2 -110.1771} C_DIS
LIN {X -97.3891,Y -37.7775,Z 102,A -162.8077,B 24.9395,C -1.796,E1 24.8509,E2 -111.591} C_DIS
LIN {X -96.4536,Y -40.1066,Z 102,A -161.395,B 24.9397,C -1.7932,E1 24.8524,E2 -113.0051} C_DIS
LIN {X -95.4988,Y -42.3317,Z 102,A -159.9863,B 24.9397,C -1.7923,E1 24.854,E2 -114.4193} C_DIS
LIN {X -94.1872,Y -45.1704,Z 102,A -158.438,B 24.9405,C -1.7815,E1 24.8558,E2 -115.9503} C_DIS
LIN {X -93.0839,Y -47.4026,Z 102,A -157.035,B 24.9407,C -1.779,E1 24.8576,E2 -117.3549} C_DIS
LIN {X -92.1259,Y -49.2423,Z 102,A -155.742,B 24.9405,C -1.7815,E1 24.8593,E2 -118.6607} C_DIS
LIN {X -90.8187,Y -51.612,Z 102,A -154.1209,B 24.9405,C -1.7825,E1 24.8615,E2 -120.2926} C_DIS
LIN {X -89.5247,Y -53.8252,Z 102,A -152.8346,B 24.941,C -1.7744,E1 24.8633,E2 -121.5662} C_DIS
LIN {X -88.1768,Y -56.0061,Z 102,A -151.4203,B 24.9412,C -1.771,E1 24.8654,E2 -122.9797} C_DIS
LIN {X -86.7758,Y -58.1532,Z 102,A -150.0779,B 24.9416,C -1.765,E1 24.8675,E2 -124.3146} C_DIS
LIN {X -85.4053,Y -60.1492,Z 102,A -148.6706,B 24.9416,C -1.7646,E1 24.8697,E2 -125.7278} C_DIS
LIN {X -83.9035,Y -62.227,Z 102,A -147.2566,B 24.9419,C -1.7614,E1 24.8721,E2 -127.141} C_DIS
LIN {X -82.3511,Y -64.2674,Z 102,A -145.7781,B 24.9419,C -1.7606,E1 24.8746,E2 -128.6247} C_DIS
LIN {X -80.658,Y -66.3787,Z 102,A -144.3508,B 24.9423,C -1.755,E1 24.8771,E2 -130.0454} C_DIS
LIN {X -79.0984,Y -68.2308,Z 102,A -143.0161,B 24.9425,C -1.7522,E1 24.8795,E2 -131.3794} C_DIS
LIN {X -77.3038,Y -70.2564,Z 102,A -141.5965,B 24.9428,C -1.7465,E1 24.8822,E2 -132.7917} C_DIS
LIN {X -74.7656,Y -72.9527,Z 102,A -139.4188,B 24.9428,C -1.7475,E1 24.8864,E2 -134.9812} C_DIS
LIN {X -72.9527,Y -74.7656,Z 102,A -138.0061,B 24.9429,C -1.7447,E1 24.8892,E2 -136.3933} C_DIS
LIN {X -71.0959,Y -76.5334,Z 102,A -136.5938,B 24.9431,C -1.7421,E1 24.8921,E2 -137.8051} C_DIS
LIN {X -69.0889,Y -78.3489,Z 102,A -135.2397,B 24.9436,C -1.7343,E1 24.8948,E2 -139.1461} C_DIS
LIN {X -67.255,Y -79.9297,Z 102,A -133.834,B 24.9436,C -1.7347,E1 24.8979,E2 -140.5581} C_DIS
LIN {X -65.1613,Y -81.6446,Z 102,A -132.3438,B 24.9438,C -1.7321,E1 24.9011,E2 -142.0479} C_DIS
LIN {X -62.9022,Y -83.3963,Z 102,A -130.8968,B 24.9442,C -1.7248,E1 24.9043,E2 -143.4828} C_DIS
LIN {X -61.0767,Y -84.7435,Z 102,A -129.5204,B 24.9441,C -1.7276,E1 24.9074,E2 -144.8706} C_DIS
LIN {X -59.0966,Y -86.137,Z 102,A -128.0315,B 24.9438,C -1.7315,E1 24.9109,E2 -146.3737} C_DIS
LIN {X -55.8861,Y -88.2538,Z 102,A -126.0712,B 24.9444,C -1.7225,E1 24.9154,E2 -148.3192} C_DIS
LIN {X -53.5807,Y -89.6713,Z 102,A -124.6537,B 24.9447,C -1.7178,E1 24.9188,E2 -149.7298} C_DIS
LIN {X -51.3639,Y -90.9592,Z 102,A -123.1716,B 24.9447,C -1.7187,E1 24.9224,E2 -151.2185} C_DIS
LIN {X -49.2423,Y -92.1259,Z 102,A -121.839,B 24.9447,C -1.7171,E1 24.9257,E2 -152.551} C_DIS
LIN {X -46.9666,Y -93.3066,Z 102,A -120.4292,B 24.9448,C -1.7155,E1 24.9292,E2 -153.9607} C_DIS
LIN {X -44.5334,Y -94.4913,Z 102,A -118.9411,B 24.945,C -1.7139,E1 24.9329,E2 -155.4488} C_DIS
LIN {X -41.1566,Y -96.0111,Z 102,A -116.8402,B 24.945,C -1.7143,E1 24.9383,E2 -157.5557} C_DIS
LIN {X -38.788,Y -96.9922,Z 102,A -115.4309,B 24.945,C -1.713,E1 24.9419,E2 -158.965} C_DIS
LIN {X -36.2621,Y -97.9637,Z 102,A -114.0799,B 24.9454,C -1.7065,E1 24.9454,E2 -160.3035} C_DIS
LIN {X -33.694,Y -98.8757,Z 102,A -112.5816,B 24.9454,C -1.7054,E1 24.9494,E2 -161.8021} C_DIS
LIN {X -31.5477,Y -99.5828,Z 102,A -111.2045,B 24.9452,C -1.7097,E1 24.9531,E2 -163.1919} C_DIS
LIN {X -28.9572,Y -100.3659,Z 102,A -109.8538,B 24.9456,C -1.7036,E1 24.9567,E2 -164.5301} C_DIS
LIN {X -26.6234,Y -101.0108,Z 102,A -108.2682,B 24.945,C -1.7127,E1 24.961,E2 -166.1399} C_DIS
LIN {X -22.6913,Y -101.9651,Z 102,A -106.2563,B 24.9456,C -1.7035,E1 24.9664,E2 -168.1326} C_DIS
LIN {X -20.3792,Y -102.4533,Z 102,A -104.8687,B 24.9454,C -1.7065,E1 24.9702,E2 -169.5291} C_DIS
LIN {X -17.7182,Y -102.9461,Z 102,A -103.5194,B 24.9458,C -1.7008,E1 24.9739,E2 -170.8661} C_DIS
LIN {X -15.3275,Y -103.3299,Z 102,A -102.0544,B 24.9455,C -1.7058,E1 24.978,E2 -172.3441} C_DIS
LIN {X -12.7871,Y -103.6749,Z 102,A -100.712,B 24.9456,C -1.703,E1 24.9817,E2 -173.681} C_DIS
LIN {X -10.097,Y -103.9706,Z 102,A -99.2989,B 24.9458,C -1.7001,E1 24.9856,E2 -175.0879} C_DIS
LIN {X -7.2793,Y -104.2049,Z 102,A -97.8803,B 24.9462,C -1.6948,E1 24.9895,E2 -176.4948} C_DIS
LIN {X -4.9652,Y -104.3416,Z 102,A -96.4858,B 24.9459,C -1.6997,E1 24.9934,E2 -177.9013} C_DIS
LIN {X -2.4211,Y -104.4317,Z 102,A -95.0805,B 24.9459,C -1.7003,E1 24.9974,E2 -179.308} C_DIS
LIN {X 0.7251,Y -104.456,Z 102,A -93.6479,B 24.9465,C -1.6891,E1 25.0013,E2 -180.7141} C_DIS
Enddeposition()
LIN {X 0.7251,Y -104.456,Z 102,A -93.6479,B 24.9465,C -1.6891,E1 25.0013,E2 -180.7141} C_DIS
Startdeposition()
$VEL.CP = VEL_PRINT
LIN {X 0.0616,Y -103.5979,Z 102,A -94.5429,B 24.9469,C -1.6835,E1 24.9988,E2 -179.806} C_DIS
LIN {X -3.9633,Y -103.5216,Z 102,A -96.6112,B 24.9465,C -1.6893,E1 24.993,E2 -177.7512} C_DIS
LIN {X -6.8958,Y -103.3666,Z 102,A -98.2999,B 24.9467,C -1.6868,E1 24.9883,E2 -176.0559} C_DIS
LIN {X -9.8126,Y -103.1309,Z 102,A -99.7881,B 24.9464,C -1.6919,E1 24.9842,E2 -174.5791} C_DIS
LIN {X -12.3402,Y -102.8591,Z 102,A -101.4055,B 24.9469,C -1.684,E1 24.9797,E2 -172.9418} C_DIS
LIN {X -16.4246,Y -102.2878,Z 102,A -103.7185,B 24.9469,C -1.6833,E1 24.9733,E2 -170.6252} C_DIS
LIN {X -19.7481,Y -101.6968,Z 102,A -105.465,B 24.9466,C -1.6886,E1 24.9685,E2 -168.8895} C_DIS
LIN {X -22.6326,Y -101.0954,Z 102,A -107.1978,B 24.9468,C -1.6854,E1 24.9637,E2 -167.1469} C_DIS
LIN {X -26.4717,Y -100.1584,Z 102,A -109.3669,B 24.9466,C -1.6873,E1 24.9579,E2 -164.9792} C_DIS
LIN {X -30.1727,Y -99.1063,Z 102,A -111.5172,B 24.9466,C -1.6879,E1 24.9521,E2 -162.8268} C_DIS
LIN {X -33.6501,Y -97.9806,Z 102,A -113.5012,B 24.9464,C -1.6909,E1 24.9469,E2 -160.8463} C_DIS
LIN {X -36.6724,Y -96.8882,Z 102,A -115.746,B 24.9474,C -1.6752,E1 24.9409,E2 -158.5594} C_DIS
LIN {X -40.1914,Y -95.4822,Z 102,A -117.1028,B 24.9455,C -1.7048,E1 24.9376,E2 -157.27} C_DIS
LIN {X -42.5759,Y -94.4431,Z 102,A -118.7189,B 24.9459,C -1.6998,E1 24.9334,E2 -155.638} C_DIS
LIN {X -45.6713,Y -92.9864,Z 102,A -120.6676,B 24.9459,C -1.6999,E1 24.9285,E2 -153.6846} C_DIS
LIN {X -48.695,Y -91.4397,Z 102,A -122.5313,B 24.9457,C -1.7029,E1 24.9239,E2 -151.8228} C_DIS
LIN {X -51.6889,Y -89.78,Z 102,A -124.4751,B 24.9457,C -1.7036,E1 24.9191,E2 -149.8752} C_DIS
LIN {X -55.3555,Y -87.5687,Z 102,A -126.9073,B 24.9455,C -1.7048,E1 24.9133,E2 -147.4382} C_DIS
LIN {X -58.6359,Y -85.4072,Z 102,A -128.8679,B 24.9448,C -1.7161,E1 24.9088,E2 -145.4979} C_DIS
LIN {X -62.4692,Y -82.6431,Z 102,A -131.5335,B 24.9446,C -1.7187,E1 24.9028,E2 -142.8291} C_DIS
LIN {X -68.613,Y -77.6198,Z 102,A -135.9163,B 24.9441,C -1.7271,E1 24.8934,E2 -138.4497} C_DIS
LIN {X -70.9868,Y -75.4524,Z 102,A -137.8784,B 24.9443,C -1.7241,E1 24.8893,E2 -136.4724} C_DIS
LIN {X -73.4708,Y -73.0366,Z 102,A -139.7451,B 24.9439,C -1.7299,E1 24.8856,E2 -134.6117} C_DIS
LIN {X -75.9269,Y -70.4816,Z 102,A -141.8019,B 24.9439,C -1.7307,E1 24.8817,E2 -132.5478} C_DIS
LIN {X -78.0048,Y -68.1722,Z 102,A -143.4938,B 24.9435,C -1.7356,E1 24.8786,E2 -130.8599} C_DIS
LIN {X -80.0457,Y -65.7663,Z 102,A -145.0728,B 24.9429,C -1.7456,E1 24.8758,E2 -129.2975} C_DIS
LIN {X -81.4862,Y -63.9711,Z 102,A -146.3501,B 24.9427,C -1.7485,E1 24.8736,E2 -128.021} C_DIS
LIN {X -83.4749,Y -61.3529,Z 102,A -148.2496,B 24.9427,C -1.75,E1 24.8704,E2 -126.1161} C_DIS
LIN {X -85.384,Y -58.6692,Z 102,A -150.9571,B 24.9443,C -1.7233,E1 24.866,E2 -123.3315} C_DIS
LIN {X -88.0747,Y -54.5453,Z 102,A -152.7063,B 24.9416,C -1.7647,E1 24.8635,E2 -121.6722} C_DIS
LIN {X -89.3549,Y -52.4214,Z 102,A -154.1539,B 24.9416,C -1.7657,E1 24.8614,E2 -120.2194} C_DIS
LIN {X -90.7621,Y -49.9484,Z 102,A -155.957,B 24.9418,C -1.7618,E1 24.8589,E2 -118.3977} C_DIS
LIN {X -93.2061,Y -45.2213,Z 102,A -158.556,B 24.9405,C -1.7821,E1 24.8557,E2 -115.8331} C_DIS
LIN {X -95.7285,Y -39.6056,Z 102,A -162.3125,B 24.9407,C -1.7794,E1 24.8514,E2 -112.0495} C_DIS
LIN {X -97.1143,Y -36.0746,Z 102,A -164.206,B 24.9398,C -1.7928,E1 24.8495,E2 -110.1771} C_DIS
LIN {X -97.8287,Y -34.0851,Z 102,A -165.4312,B 24.9397,C -1.7943,E1 24.8484,E2 -108.9487} C_DIS
LIN {X -98.9705,Y -30.611,Z 102,A -167.5469,B 24.9395,C -1.7971,E1 24.8466,E2 -106.8276} C_DIS
LIN {X -99.877,Y -27.5146,Z 102,A -169.1919,B 24.9388,C -1.8074,E1 24.8453,E2 -105.1975} C_DIS
LIN {X -100.5142,Y -25.0877,Z 102,A -171.7501,B 24.9412,C -1.7711,E1 24.8436,E2 -102.5379} C_DIS
LIN {X -101.7263,Y -19.5947,Z 102,A -174.9217,B 24.9407,C -1.7788,E1 24.8419,E2 -99.3658} C_DIS
LIN {X -102.6742,Y -13.8003,Z 102,A -177.1279,B 24.9376,C -1.8249,E1 24.8411,E2 -97.2564} C_DIS
LIN {X -103.0659,Y -10.474,Z 102,A -178.8109,B 24.9368,C -1.8367,E1 24.8405,E2 -95.5914} C_DIS
LIN {X -103.3218,Y -7.558,Z 102,A 179.2885,B 24.9371,C -1.832,E1 24.8401,E2 -93.6683} C_DIS
LIN {X -103.5296,Y -3.7636,Z 102,A 177.1337,B 24.9368,C -1.8369,E1 24.8398,E2 -91.5123} C_DIS
LIN {X -103.5959,Y -0.381,Z 102,A 175.4544,B 24.9359,C -1.8496,E1 24.8398,E2 -89.8531} C_DIS
LIN {X -103.5793,Y 1.8742,Z 102,A 174.1185,B 24.9359,C -1.8506,E1 24.8398,E2 -88.5114} C_DIS
LIN {X -103.4441,Y 5.6139,Z 102,A 172.032,B 24.9354,C -1.8567,E1 24.8401,E2 -86.4269} C_DIS
LIN {X -103.1893,Y 9.1802,Z 102,A 170.1435,B 24.9347,C -1.8661,E1 24.8405,E2 -84.5496} C_DIS
LIN {X -102.7634,Y 13.112,Z 102,A 168.1639,B 24.9337,C -1.8804,E1 24.8411,E2 -82.5923} C_DIS
LIN {X -101.7197,Y 19.6291,Z 102,A 164.6127,B 24.9326,C -1.8956,E1 24.8427,E2 -79.0561} C_DIS
LIN {X -100.343,Y 25.7582,Z 102,A 160.6859,B 24.933,C -1.8908,E1 24.8452,E2 -75.0949} C_DIS
LIN {X -98.9716,Y 30.6074,Z 102,A 157.4661,B 24.9334,C -1.8846,E1 24.8477,E2 -71.8417} C_DIS
LIN {X -97.9461,Y 33.7505,Z 102,A 156.0705,B 24.9319,C -1.9053,E1 24.8489,E2 -70.4875} C_DIS
LIN {X -97.1589,Y 35.9524,Z 102,A 154.8143,B 24.9316,C -1.9106,E1 24.8501,E2 -69.2368} C_DIS
LIN {X -95.9401,Y 39.0858,Z 102,A 152.7687,B 24.9316,C -1.9098,E1 24.8522,E2 -67.178} C_DIS
LIN {X -94.6552,Y 42.105,Z 102,A 150.9293,B 24.9313,C -1.9145,E1 24.8543,E2 -65.3395} C_DIS
LIN {X -93.1708,Y 45.2946,Z 102,A 148.0576,B 24.9332,C -1.8884,E1 24.8579,E2 -62.39} C_DIS
LIN {X -90.6043,Y 50.231,Z 102,A 145.9735,B 24.93,C -1.9316,E1 24.8606,E2 -60.3981} C_DIS
LIN {X -88.8373,Y 53.2961,Z 102,A 144.1149,B 24.9294,C -1.9407,E1 24.8632,E2 -58.5514} C_DIS
LIN {X -87.7447,Y 55.0737,Z 102,A 142.7957,B 24.9296,C -1.9382,E1 24.8651,E2 -57.2196} C_DIS
LIN {X -85.2576,Y 58.8511,Z 102,A 140.5661,B 24.9284,C -1.9547,E1 24.8685,E2 -55.0182} C_DIS
LIN {X -81.7929,Y 63.5791,Z 102,A 137.1704,B 24.9281,C -1.958,E1 24.8742,E2 -51.614} C_DIS
LIN {X -80.4299,Y 65.2934,Z 102,A 135.8944,B 24.9281,C -1.959,E1 24.8764,E2 -50.3343} C_DIS
LIN {X -78.9367,Y 67.091,Z 102,A 134.5273,B 24.928,C -1.9597,E1 24.8789,E2 -48.9626} C_DIS
LIN {X -76.6566,Y 69.6864,Z 102,A 132.5861,B 24.9277,C -1.9634,E1 24.8825,E2 -47.0217} C_DIS
LIN {X -74.3416,Y 72.1501,Z 102,A 130.8382,B 24.9271,C -1.9724,E1 24.8858,E2 -45.2875} C_DIS
LIN {X -72.246,Y 74.2492,Z 102,A 129.0735,B 24.9271,C -1.9719,E1 24.8894,E2 -43.5143} C_DIS
LIN {X -69.8233,Y 76.531,Z 102,A 127.2324,B 24.9268,C -1.9762,E1 24.8931,E2 -41.6759} C_DIS
LIN {X -67.1502,Y 78.8863,Z 102,A 125.2757,B 24.9264,C -1.9812,E1 24.8972,E2 -39.7233} C_DIS
LIN {X -65.0623,Y 80.6172,Z 102,A 123.8548,B 24.926,C -1.9873,E1 24.9003,E2 -38.3116} C_DIS
LIN {X -62.4934,Y 82.625,Z 102,A 121.8736,B 24.9261,C -1.9847,E1 24.9047,E2 -36.3171} C_DIS
LIN {X -59.4645,Y 84.8312,Z 102,A 119.5691,B 24.9264,C -1.9807,E1 24.91,E2 -33.995} C_DIS
LIN {X -56.527,Y 86.8173,Z 102,A 117.9864,B 24.9252,C -1.998,E1 24.9136,E2 -32.4483} C_DIS
LIN {X -53.8658,Y 88.4911,Z 102,A 116.2342,B 24.9249,C -2.0008,E1 24.9178,E2 -30.6972} C_DIS
LIN {X -51.0271,Y 90.1598,Z 102,A 114.0548,B 24.9257,C -1.9911,E1 24.9231,E2 -28.4884} C_DIS
LIN {X -47.1748,Y 92.2319,Z 102,A 111.9699,B 24.9245,C -2.0072,E1 24.9282,E2 -26.4361} C_DIS
LIN {X -44.6475,Y 93.4818,Z 102,A 110.2171,B 24.9248,C -2.0027,E1 24.9326,E2 -24.6679} C_DIS
LIN {X -41.2373,Y 95.0353,Z 102,A 107.6646,B 24.9259,C -1.9884,E1 24.9392,E2 -22.0755} C_DIS
LIN {X -37.6043,Y 96.5308,Z 102,A 106.189,B 24.9237,C -2.0167,E1 24.9429,E2 -20.6638} C_DIS
LIN {X -35.1013,Y 97.4693,Z 102,A 104.4822,B 24.9242,C -2.0102,E1 24.9474,E2 -18.9383} C_DIS
LIN {X -30.657,Y 98.9563,Z 102,A 102.2341,B 24.923,C -2.0259,E1 24.9533,E2 -16.7234} C_DIS
LIN {X -27.9042,Y 99.7681,Z 102,A 100.3025,B 24.9239,C -2.015,E1 24.9586,E2 -14.7625} C_DIS
LIN {X -24.0988,Y 100.7554,Z 102,A 97.9464,B 24.9242,C -2.0104,E1 24.965,E2 -12.3922} C_DIS
LIN {X -18.8594,Y 101.8666,Z 102,A 95.1469,B 24.9236,C -2.0188,E1 24.9726,E2 -9.6096} C_DIS
LIN {X -15.2213,Y 102.4738,Z 102,A 93.082,B 24.9236,C -2.0193,E1 24.9783,E2 -7.544} C_DIS
LIN {X -11.925,Y 102.9077,Z 102,A 91.411,B 24.923,C -2.0267,E1 24.9829,E2 -5.8893} C_DIS
LIN {X -8.512,Y 103.2463,Z 102,A 89.4882,B 24.923,C -2.0267,E1 24.9882,E2 -3.9655} C_DIS
LIN {X -5.6558,Y 103.4418,Z 102,A 87.8937,B 24.923,C -2.0268,E1 24.9927,E2 -2.3709} C_DIS
LIN {X -1.783,Y 103.581,Z 102,A 85.8416,B 24.9227,C -2.0309,E1 24.9984,E2 -0.3281} C_DIS
LIN {X 1.3489,Y 103.589,Z 102,A 84.099,B 24.9227,C -2.0308,E1 25.0033,E2 1.4146} C_DIS
LIN {X 4.7753,Y 103.4867,Z 102,A 82.1505,B 24.9228,C -2.029,E1 25.0087,E2 3.3669} C_DIS
LIN {X 7.6009,Y 103.3189,Z 102,A 80.4097,B 24.9233,C -2.0222,E1 25.0136,E2 5.1228} C_DIS
LIN {X 10.7629,Y 103.0357,Z 102,A 78.7351,B 24.9231,C -2.0251,E1 25.0182,E2 6.7896} C_DIS
LIN {X 13.7852,Y 102.6761,Z 102,A 76.9826,B 24.9233,C -2.0221,E1 25.0231,E2 8.5478} C_DIS
LIN {X 17.0678,Y 102.1806,Z 102,A 75.2493,B 24.9231,C -2.0255,E1 25.0278,E2 10.2714} C_DIS
LIN {X 19.9657,Y 101.6549,Z 102,A 73.5284,B 24.9234,C -2.0213,E1 25.0326,E2 12.0003} C_DIS
LIN {X 23.7166,Y 100.8458,Z 102,A 71.4088,B 24.9234,C -2.0203,E1 25.0384,E2 14.1194} C_DIS
LIN {X 27.3359,Y 99.9252,Z 102,A 69.3474,B 24.9236,C -2.0191,E1 25.0439,E2 16.1804} C_DIS
LIN {X 30.7785,Y 98.9186,Z 102,A 67.4912,B 24.9233,C -2.0226,E1 25.0489,E2 18.025} C_DIS
LIN {X 33.9024,Y 97.8928,Z 102,A 65.0092,B 24.9253,C -1.9954,E1 25.0556,E2 20.5665} C_DIS
LIN {X 37.8077,Y 96.4509,Z 102,A 63.4269,B 24.9234,C -2.0211,E1 25.0595,E2 22.0846} C_DIS
LIN {X 40.6038,Y 95.3084,Z 102,A 61.6813,B 24.9238,C -2.0163,E1 25.064,E2 23.8373} C_DIS
LIN {X 43.7918,Y 93.8855,Z 102,A 59.7611,B 24.9239,C -2.0145,E1 25.0689,E2 25.757} C_DIS
LIN {X 47.132,Y 92.2538,Z 102,A 57.7037,B 24.9241,C -2.0119,E1 25.0741,E2 27.8151} C_DIS
LIN {X 49.6506,Y 90.9236,Z 102,A 56.0984,B 24.9244,C -2.0086,E1 25.078,E2 29.4236} C_DIS
LIN {X 52.6496,Y 89.22,Z 102,A 54.2889,B 24.9243,C -2.0097,E1 25.0824,E2 31.225} C_DIS
LIN {X 55.417,Y 87.5302,Z 102,A 52.5516,B 24.9243,C -2.0091,E1 25.0865,E2 32.9581} C_DIS
LIN {X 58.6663,Y 85.3861,Z 102,A 50.2754,B 24.9249,C -2.0007,E1 25.0918,E2 35.2466} C_DIS
LIN {X 61.6833,Y 83.2329,Z 102,A 48.2716,B 24.9251,C -1.999,E1 25.0963,E2 37.2474} C_DIS
LIN {X 64.1922,Y 81.3115,Z 102,A 46.1838,B 24.9263,C -1.9823,E1 25.101,E2 39.367} C_DIS
LIN {X 67.3879,Y 78.6838,Z 102,A 44.3402,B 24.9253,C -1.9957,E1 25.1048,E2 41.1719} C_DIS
LIN {X 69.835,Y 76.5202,Z 102,A 42.4902,B 24.9257,C -1.9903,E1 25.1087,E2 43.0272} C_DIS
LIN {X 72.748,Y 73.7559,Z 102,A 38.8864,B 24.9301,C -1.9306,E1 25.1161,E2 46.7569} C_DIS
LIN {X 77.5985,Y 68.6371,Z 102,A 36.455,B 24.9265,C -1.9804,E1 25.1205,E2 49.0597} C_DIS
LIN {X 79.9073,Y 65.9329,Z 102,A 34.497,B 24.9268,C -1.9762,E1 25.124,E2 51.0188} C_DIS
LIN {X 82.3442,Y 62.8637,Z 102,A 32.3067,B 24.9272,C -1.97,E1 25.1278,E2 53.2133} C_DIS
LIN {X 84.5178,Y 59.9086,Z 102,A 30.2677,B 24.9276,C -1.9646,E1 25.1311,E2 55.2554} C_DIS
LIN {X 86.8185,Y 56.5252,Z 102,A 28.0844,B 24.9278,C -1.962,E1 25.1345,E2 57.4339} C_DIS
LIN {X 88.8592,Y 53.2601,Z 102,A 25.7403,B 24.9289,C -1.9476,E1 25.1379,E2 59.8002} C_DIS
LIN {X 90.7213,Y 50.0208,Z 102,A 23.7087,B 24.9292,C -1.9434,E1 25.1407,E2 61.8311} C_DIS
LIN {X 92.433,Y 46.7815,Z 102,A 21.9096,B 24.9289,C -1.9472,E1 25.143,E2 63.6119} C_DIS
LIN {X 93.6754,Y 44.243,Z 102,A 20.3588,B 24.9292,C -1.9432,E1 25.1449,E2 65.1635} C_DIS
LIN {X 94.7465,Y 41.8998,Z 102,A 18.9596,B 24.9294,C -1.9402,E1 25.1465,E2 66.5622} C_DIS
LIN {X 96.198,Y 38.4515,Z 102,A 16.8671,B 24.9299,C -1.9333,E1 25.1487,E2 68.6597} C_DIS
LIN {X 97.7571,Y 34.2891,Z 102,A 14.4005,B 24.9305,C -1.9257,E1 25.1511,E2 71.1304} C_DIS
LIN {X 98.5737,Y 31.8655,Z 102,A 13.0142,B 24.9307,C -1.9226,E1 25.1523,E2 72.5161} C_DIS
LIN {X 99.4541,Y 29.0053,Z 102,A 11.3242,B 24.9312,C -1.9161,E1 25.1537,E2 74.2118} C_DIS
LIN {X 100.6176,Y 24.6637,Z 102,A 8.8546,B 24.9317,C -1.9092,E1 25.1555,E2 76.6835} C_DIS
LIN {X 101.3698,Y 21.3697,Z 102,A 6.8331,B 24.9325,C -1.897,E1 25.1567,E2 78.722} C_DIS
LIN {X 102.1038,Y 17.5242,Z 102,A 4.888,B 24.9324,C -1.8994,E1 25.1576,E2 80.6501} C_DIS
LIN {X 102.6157,Y 14.2242,Z 102,A 2.8418,B 24.9334,C -1.8852,E1 25.1585,E2 82.7176} C_DIS
LIN {X 103.1012,Y 10.1347,Z 102,A 0.7864,B 24.9332,C -1.8872,E1 25.1591,E2 84.7562} C_DIS
LIN {X 103.3639,Y 6.9352,Z 102,A -0.9626,B 24.9336,C -1.8826,E1 25.1595,E2 86.5056} C_DIS
LIN {X 103.5281,Y 3.8132,Z 102,A -2.9092,B 24.9346,C -1.868,E1 25.1597,E2 88.4751} C_DIS
LIN {X 103.597,Y -0.2107,Z 102,A -4.876,B 24.9343,C -1.8716,E1 25.1597,E2 90.4217} C_DIS
LIN {X 103.5696,Y -2.4061,Z 102,A -6.1115,B 24.9347,C -1.8668,E1 25.1597,E2 91.6612} C_DIS
LIN {X 103.4327,Y -5.8209,Z 102,A -7.9403,B 24.9349,C -1.8633,E1 25.1595,E2 93.4875} C_DIS
LIN {X 103.225,Y -8.7789,Z 102,A -9.7881,B 24.9359,C -1.8492,E1 25.1591,E2 95.3574} C_DIS
LIN {X 102.9088,Y -11.9162,Z 102,A -11.4519,B 24.9361,C -1.847,E1 25.1586,E2 97.0167} C_DIS
LIN {X 102.5324,Y -14.8106,Z 102,A -13.1075,B 24.9365,C -1.84,E1 25.1579,E2 98.6789} C_DIS
LIN {X 101.8441,Y -18.9831,Z 102,A -15.2565,B 24.9365,C -1.8404,E1 25.1569,E2 100.8144} C_DIS
LIN {X 101.3113,Y -21.6429,Z 102,A -16.661,B 24.9365,C -1.8396,E1 25.1561,E2 102.2126} C_DIS
LIN {X 100.673,Y -24.4367,Z 102,A -18.3841,B 24.9373,C -1.8288,E1 25.155,E2 103.9512} C_DIS
LIN {X 99.9716,Y -27.1641,Z 102,A -20.0067,B 24.9378,C -1.8211,E1 25.1539,E2 105.5826} C_DIS
LIN {X 98.8962,Y -30.8509,Z 102,A -22.163,B 24.9384,C -1.8131,E1 25.1521,E2 107.7455} C_DIS
LIN {X 97.7121,Y -34.4173,Z 102,A -24.0873,B 24.9384,C -1.813,E1 25.1504,E2 109.6593} C_DIS
LIN {X 96.3933,Y -37.9542,Z 102,A -26.0963,B 24.9386,C -1.8098,E1 25.1484,E2 111.6645} C_DIS
LIN {X 95.1884,Y -40.8861,Z 102,A -28.0954,B 24.9397,C -1.7942,E1 25.1462,E2 113.6896} C_DIS
LIN {X 93.5675,Y -44.4693,Z 102,A -30.1964,B 24.9399,C -1.7907,E1 25.1438,E2 115.7874} C_DIS
LIN {X 91.8677,Y -47.8813,Z 102,A -32.3164,B 24.9404,C -1.7839,E1 25.1411,E2 117.9121} C_DIS
LIN {X 90.4539,Y -50.5003,Z 102,A -33.8291,B 24.9404,C -1.7846,E1 25.139,E2 119.4152} C_DIS
LIN {X 88.1512,Y -54.4229,Z 102,A -36.2139,B 24.9404,C -1.7827,E1 25.1357,E2 121.7922} C_DIS
LIN {X 86.8875,Y -56.418,Z 102,A -37.753,B 24.9413,C -1.7694,E1 25.1333,E2 123.3552} C_DIS
LIN {X 84.743,Y -59.5914,Z 102,A -40.9188,B 24.9445,C -1.7206,E1 25.1281,E2 126.6204} C_DIS
LIN {X 81.0047,Y -64.5804,Z 102,A -44.1403,B 24.9445,C -1.7206,E1 25.1225,E2 129.8269} C_DIS
LIN {X 77.503,Y -68.7437,Z 102,A -46.3132,B 24.9428,C -1.7469,E1 25.1186,E2 131.9279} C_DIS
LIN {X 73.6632,Y -72.8418,Z 102,A -49.1449,B 24.9426,C -1.7505,E1 25.1132,E2 134.7391} C_DIS
LIN {X 71.5748,Y -74.8962,Z 102,A -50.8077,B 24.9429,C -1.7448,E1 25.1099,E2 136.4084} C_DIS
LIN {X 69.4359,Y -76.8834,Z 102,A -52.6689,B 24.9439,C -1.7309,E1 25.106,E2 138.2948} C_DIS
LIN {X 64.7516,Y -80.869,Z 102,A -55.7674,B 24.9435,C -1.7356,E1 25.0994,E2 141.3702} C_DIS
LIN {X 60.536,Y -84.0701,Z 102,A -59.4262,B 24.9459,C -1.6998,E1 25.091,E2 145.1005} C_DIS
LIN {X 57.1274,Y -86.4215,Z 102,A -61.0961,B 24.9445,C -1.7203,E1 25.0873,E2 146.7164} C_DIS
LIN {X 54.4502,Y -88.1342,Z 102,A -63.0269,B 24.9452,C -1.7099,E1 25.0826,E2 148.6656} C_DIS
LIN {X 51.7479,Y -89.7461,Z 102,A -64.5986,B 24.945,C -1.7136,E1 25.0789,E2 150.2239} C_DIS
LIN {X 48.9226,Y -91.3184,Z 102,A -66.2481,B 24.9448,C -1.716,E1 25.0749,E2 151.8628} C_DIS
LIN {X 45.2197,Y -93.2069,Z 102,A -68.4554,B 24.9448,C -1.716,E1 25.0694,E2 154.0643} C_DIS
LIN {X 42.4863,Y -94.4834,Z 102,A -70.3167,B 24.9455,C -1.7056,E1 25.0646,E2 155.9455} C_DIS
LIN {X 39.6749,Y -95.6996,Z 102,A -71.9161,B 24.9455,C -1.7068,E1 25.0605,E2 157.538} C_DIS
LIN {X 36.7389,Y -96.863,Z 102,A -73.7801,B 24.9459,C -1.6998,E1 25.0556,E2 159.4147} C_DIS
LIN {X 32.3448,Y -98.4187,Z 102,A -76.2597,B 24.9459,C -1.7004,E1 25.0491,E2 161.888} C_DIS
LIN {X 29.131,Y -99.4168,Z 102,A -78.1174,B 24.9459,C -1.6984,E1 25.0441,E2 163.747} C_DIS
LIN {X 26.1548,Y -100.241,Z 102,A -79.6222,B 24.9455,C -1.7046,E1 25.0401,E2 165.2347} C_DIS
LIN {X 22.3181,Y -101.164,Z 102,A -82.0182,B 24.9462,C -1.6941,E1 25.0335,E2 167.6523} C_DIS
LIN {X 19.3436,Y -101.7746,Z 102,A -83.6413,B 24.9462,C -1.6949,E1 25.0291,E2 169.2716} C_DIS
LIN {X 16.0044,Y -102.3527,Z 102,A -85.578,B 24.9464,C -1.691,E1 25.0238,E2 171.2155} C_DIS
LIN {X 12.6289,Y -102.8253,Z 102,A -87.5083,B 24.9466,C -1.688,E1 25.0184,E2 173.1513} C_DIS
LIN {X 9.4897,Y -103.1607,Z 102,A -89.2591,B 24.9466,C -1.6868,E1 25.0135,E2 174.9037} C_DIS
LIN {X 6.4169,Y -103.3989,Z 102,A -90.8159,B 24.9464,C -1.6918,E1 25.0092,E2 176.4481} C_DIS
LIN {X 3.8132,Y -103.5281,Z 102,A -92.2477,B 24.9464,C -1.6916,E1 25.0052,E2 177.8798} C_DIS
LIN {X 0.7183,Y -103.5927,Z 102,A -93.5911,B 24.9455,C -1.7056,E1 25.0016,E2 179.19} C_DIS
Enddeposition()
LIN {X 0.7183,Y -103.5927,Z 102,A -93.5911,B 24.9455,C -1.7056,E1 25.0016,E2 179.19} C_DIS
Startdeposition()
$VEL.CP = VEL_PRINT
LIN {X 1.3173,Y -102.7272,Z 102,A -92.8143,B 24.9434,C -1.7379,E1 25.004,E2 178.3367} C_DIS
LIN {X 6.6224,Y -102.5209,Z 102,A -90.1974,B 24.9442,C -1.7256,E1 25.0112,E2 175.7499} C_DIS
LIN {X 9.28,Y -102.3142,Z 102,A -88.4697,B 24.9435,C -1.7357,E1 25.016,E2 173.999} C_DIS
LIN {X 12.4707,Y -101.9757,Z 102,A -86.6584,B 24.9435,C -1.7377,E1 25.0211,E2 172.1844} C_DIS
LIN {X 16.5422,Y -101.3943,Z 102,A -84.4346,B 24.9435,C -1.7365,E1 25.0272,E2 169.9653} C_DIS
LIN {X 20.8743,Y -100.5912,Z 102,A -82.0063,B 24.9435,C -1.7375,E1 25.0339,E2 167.5377} C_DIS
LIN {X 23.7599,Y -99.9506,Z 102,A -80.3209,B 24.9432,C -1.7405,E1 25.0385,E2 165.8475} C_DIS
LIN {X 26.6569,Y -99.2155,Z 102,A -78.6086,B 24.943,C -1.744,E1 25.0431,E2 164.1294} C_DIS
LIN {X 30.1377,Y -98.2146,Z 102,A -75.919,B 24.9411,C -1.7733,E1 25.0505,E2 161.3752} C_DIS
LIN {X 34.2952,Y -96.8412,Z 102,A -74.0783,B 24.9425,C -1.7521,E1 25.0552,E2 159.5884} C_DIS
LIN {X 38.6967,Y -95.1675,Z 102,A -71.637,B 24.9427,C -1.7483,E1 25.0615,E2 157.1614} C_DIS
LIN {X 41.3578,Y -94.0422,Z 102,A -70.0367,B 24.9426,C -1.7503,E1 25.0656,E2 155.5604} C_DIS
LIN {X 44.0383,Y -92.8179,Z 102,A -68.4785,B 24.9426,C -1.7494,E1 25.0695,E2 154.0081} C_DIS
LIN {X 49.7046,Y -89.9107,Z 102,A -63.941,B 24.9396,C -1.7957,E1 25.0809,E2 149.3741} C_DIS
LIN {X 53.9806,Y -87.4109,Z 102,A -62.0504,B 24.9416,C -1.7651,E1 25.0853,E2 147.5618} C_DIS
LIN {X 57.0101,Y -85.466,Z 102,A -59.5535,B 24.94,C -1.7891,E1 25.0912,E2 145.0164} C_DIS
LIN {X 59.831,Y -83.514,Z 102,A -57.5256,B 24.9394,C -1.7978,E1 25.0958,E2 142.9751} C_DIS
LIN {X 63.0617,Y -81.1031,Z 102,A -55.8023,B 24.9406,C -1.781,E1 25.0995,E2 141.2979} C_DIS
LIN {X 66.8285,Y -78.0265,Z 102,A -53.0728,B 24.9401,C -1.7878,E1 25.1054,E2 138.5628} C_DIS
LIN {X 70.1882,Y -75.0181,Z 102,A -50.2342,B 24.9388,C -1.8071,E1 25.1113,E2 135.69} C_DIS
LIN {X 72.7288,Y -72.5608,Z 102,A -48.2702,B 24.9385,C -1.8116,E1 25.1152,E2 133.7238} C_DIS
LIN {X 75.012,Y -70.1949,Z 102,A -46.7313,B 24.939,C -1.8039,E1 25.1181,E2 132.2096} C_DIS
LIN {X 78.0127,Y -66.8452,Z 102,A -44.1745,B 24.9384,C -1.8124,E1 25.1228,E2 129.6443} C_DIS
LIN {X 80.6732,Y -63.6093,Z 102,A -42.255,B 24.9392,C -1.8013,E1 25.1261,E2 127.7599} C_DIS
LIN {X 83.9993,Y -59.1506,Z 102,A -39.0335,B 24.9383,C -1.8147,E1 25.1315,E2 124.5224} C_DIS
LIN {X 85.5812,Y -56.8354,Z 102,A -37.2242,B 24.9373,C -1.8293,E1 25.1343,E2 122.6876} C_DIS
LIN {X 87.445,Y -53.926,Z 102,A -34.9503,B 24.9359,C -1.8494,E1 25.1377,E2 120.3778} C_DIS
LIN {X 89.4279,Y -50.5691,Z 102,A -33.3017,B 24.937,C -1.8336,E1 25.1399,E2 118.775} C_DIS
LIN {X 91.6064,Y -46.5041,Z 102,A -30.7056,B 24.9364,C -1.8423,E1 25.1433,E2 116.1722} C_DIS
LIN {X 93.1128,Y -43.4086,Z 102,A -28.993,B 24.9366,C -1.8394,E1 25.1453,E2 114.4756} C_DIS
LIN {X 94.2169,Y -40.9569,Z 102,A -27.467,B 24.9362,C -1.8451,E1 25.1471,E2 112.9446} C_DIS
LIN {X 96.3442,Y -35.6698,Z 102,A -24.2484,B 24.9354,C -1.8565,E1 25.1504,E2 109.7168} C_DIS
LIN {X 98.198,Y -30.1911,Z 102,A -20.9521,B 24.9345,C -1.8696,E1 25.1532,E2 106.4083} C_DIS
LIN {X 99.2668,Y -26.4672,Z 102,A -18.8735,B 24.9342,C -1.873,E1 25.1548,E2 104.3336} C_DIS
LIN {X 100.1407,Y -22.9381,Z 102,A -16.4942,B 24.9327,C -1.8943,E1 25.1563,E2 101.9179} C_DIS
LIN {X 100.8132,Y -19.7766,Z 102,A -15.1308,B 24.9336,C -1.8815,E1 25.157,E2 100.5924} C_DIS
LIN {X 101.519,Y -15.7541,Z 102,A -12.8836,B 24.9332,C -1.8876,E1 25.1581,E2 98.3441} C_DIS
LIN {X 101.939,Y -12.764,Z 102,A -11.1676,B 24.9327,C -1.8944,E1 25.1587,E2 96.6223} C_DIS
LIN {X 102.2714,Y -9.7438,Z 102,A -9.4011,B 24.9321,C -1.9029,E1 25.1592,E2 94.8462} C_DIS
LIN {X 102.5504,Y -6.1594,Z 102,A -7.3884,B 24.9316,C -1.9097,E1 25.1596,E2 92.8294} C_DIS
LIN {X 102.7075,Y -2.3912,Z 102,A -5.3217,B 24.9313,C -1.9149,E1 25.1598,E2 90.7626} C_DIS
LIN {X 102.7279,Y 1.279,Z 102,A -3.1623,B 24.9304,C -1.9263,E1 25.1598,E2 88.5893} C_DIS
LIN {X 102.5964,Y 5.3275,Z 102,A -1.1012,B 24.9305,C -1.9252,E1 25.1595,E2 86.5429} C_DIS
LIN {X 102.3516,Y 8.8745,Z 102,A 0.9281,B 24.9299,C -1.9335,E1 25.159,E2 84.5061} C_DIS
LIN {X 101.9675,Y 12.5409,Z 102,A 2.9514,B 24.9295,C -1.9387,E1 25.1584,E2 82.4826} C_DIS
LIN {X 101.504,Y 15.8509,Z 102,A 4.9866,B 24.9286,C -1.9518,E1 25.1575,E2 80.4284} C_DIS
LIN {X 100.6776,Y 20.4539,Z 102,A 7.3327,B 24.9288,C -1.949,E1 25.1563,E2 78.1027} C_DIS
LIN {X 99.598,Y 25.1928,Z 102,A 11.027,B 24.9251,C -1.9987,E1 25.1538,E2 74.3124} C_DIS
LIN {X 98.0793,Y 30.574,Z 102,A 12.9387,B 24.9282,C -1.9575,E1 25.1524,E2 72.5089} C_DIS
LIN {X 95.9035,Y 36.838,Z 102,A 16.8329,B 24.9268,C -1.9765,E1 25.1487,E2 68.5916} C_DIS
LIN {X 94.693,Y 39.8439,Z 102,A 18.5337,B 24.9267,C -1.9774,E1 25.1469,E2 66.8981} C_DIS
LIN {X 92.6889,Y 44.3069,Z 102,A 21.3242,B 24.9259,C -1.9877,E1 25.1436,E2 64.0985} C_DIS
LIN {X 91.0845,Y 47.5191,Z 102,A 23.3451,B 24.9254,C -1.994,E1 25.141,E2 62.0734} C_DIS
LIN {X 88.1196,Y 52.8169,Z 102,A 26.7676,B 24.9247,C -2.0046,E1 25.1363,E2 58.6435} C_DIS
LIN {X 85.997,Y 56.2048,Z 102,A 29.7204,B 24.9219,C -2.0403,E1 25.1317,E2 55.6211} C_DIS
LIN {X 83.1724,Y 60.3064,Z 102,A 31.5703,B 24.9243,C -2.009,E1 25.1288,E2 53.8543} C_DIS
LIN {X 79.6711,Y 64.8603,Z 102,A 34.9025,B 24.9233,C -2.022,E1 25.1231,E2 50.5071} C_DIS
LIN {X 76.9418,Y 68.078,Z 102,A 37.892,B 24.9209,C -2.0534,E1 25.1175,E2 47.4567} C_DIS
LIN {X 73.9456,Y 71.3185,Z 102,A 39.7323,B 24.9225,C -2.0334,E1 25.114,E2 45.6716} C_DIS
LIN {X 71.3934,Y 73.8734,Z 102,A 41.7632,B 24.9221,C -2.0384,E1 25.1099,E2 43.6376} C_DIS
LIN {X 68.672,Y 76.4099,Z 102,A 43.7476,B 24.9221,C -2.0389,E1 25.1059,E2 41.6599} C_DIS
LIN {X 65.8017,Y 78.8952,Z 102,A 47.0302,B 24.9181,C -2.0904,E1 25.0986,E2 38.2682} C_DIS
LIN {X 60.6903,Y 82.8913,Z 102,A 49.3863,B 24.9215,C -2.0455,E1 25.0936,E2 36.0266} C_DIS
LIN {X 55.9211,Y 86.1822,Z 102,A 52.7039,B 24.9209,C -2.0542,E1 25.0859,E2 32.6997} C_DIS
LIN {X 52.7242,Y 88.1744,Z 102,A 54.6416,B 24.9211,C -2.0509,E1 25.0813,E2 30.7759} C_DIS
LIN {X 48.8491,Y 90.3774,Z 102,A 57.2145,B 24.9206,C -2.0579,E1 25.075,E2 28.1942} C_DIS
LIN {X 45.5796,Y 92.0695,Z 102,A 59.216,B 24.9206,C -2.0584,E1 25.07,E2 26.1968} C_DIS
LIN {X 43.0654,Y 93.2725,Z 102,A 61.1191,B 24.9193,C -2.0741,E1 25.0651,E2 24.2615} C_DIS
LIN {X 38.6437,Y 95.1891,Z 102,A 63.5263,B 24.92,C -2.0658,E1 25.059,E2 21.8794} C_DIS
LIN {X 34.6067,Y 96.7319,Z 102,A 66.6079,B 24.9177,C -2.0945,E1 25.0508,E2 18.7363} C_DIS
LIN {X 30.4239,Y 98.1258,Z 102,A 68.2905,B 24.92,C -2.066,E1 25.0465,E2 17.1245} C_DIS
LIN {X 28.1884,Y 98.7914,Z 102,A 69.8812,B 24.919,C -2.0782,E1 25.0421,E2 15.5075} C_DIS
LIN {X 23.9467,Y 99.905,Z 102,A 72.1639,B 24.9194,C -2.0732,E1 25.036,E2 13.2399} C_DIS
LIN {X 20.6899,Y 100.6291,Z 102,A 73.9432,B 24.9196,C -2.071,E1 25.0311,E2 11.4682} C_DIS
LIN {X 17.6845,Y 101.2018,Z 102,A 75.9067,B 24.9187,C -2.0816,E1 25.0257,E2 9.4818} C_DIS
LIN {X 12.6975,Y 101.9476,Z 102,A 78.5142,B 24.9193,C -2.0744,E1 25.0185,E2 6.8936} C_DIS
LIN {X 10.0113,Y 102.2467,Z 102,A 80.0529,B 24.9192,C -2.0757,E1 25.0142,E2 5.3526} C_DIS
LIN {X 6.3656,Y 102.5382,Z 102,A 82.0857,B 24.9192,C -2.0755,E1 25.0086,E2 3.3212} C_DIS
LIN {X 2.9806,Y 102.691,Z 102,A 83.8836,B 24.9195,C -2.0719,E1 25.0036,E2 1.5324} C_DIS
LIN {X -0.6802,Y 102.7318,Z 102,A 85.8962,B 24.9196,C -2.0704,E1 24.998,E2 -0.4766} C_DIS
LIN {X -4.0125,Y 102.6565,Z 102,A 87.8345,B 24.9194,C -2.0729,E1 24.9925,E2 -2.4209} C_DIS
LIN {X -7.6431,Y 102.4504,Z 102,A 90.1698,B 24.9186,C -2.0836,E1 24.986,E2 -4.7827} C_DIS
LIN {X -11.9029,Y 102.0422,Z 102,A 92.1475,B 24.9199,C -2.067,E1 24.9806,E2 -6.722} C_DIS
LIN {X -15.115,Y 101.6178,Z 102,A 93.9008,B 24.9201,C -2.0638,E1 24.9758,E2 -8.4691} C_DIS
LIN {X -19.8755,Y 100.7942,Z 102,A 96.6689,B 24.9201,C -2.0645,E1 24.9681,E2 -11.2417} C_DIS
LIN {X -26.7994,Y 99.177,Z 102,A 100.6558,B 24.9203,C -2.0614,E1 24.9573,E2 -15.2269} C_DIS
LIN {X -33.3544,Y 97.1704,Z 102,A 104.5959,B 24.9203,C -2.0613,E1 24.9468,E2 -19.1735} C_DIS
LIN {X -36.6577,Y 95.9718,Z 102,A 106.3547,B 24.9211,C -2.0513,E1 24.9423,E2 -20.9123} C_DIS
LIN {X -40.3671,Y 94.4721,Z 102,A 109.0162,B 24.9201,C -2.0639,E1 24.9353,E2 -23.6098} C_DIS
LIN {X -46.0757,Y 91.8236,Z 102,A 113.17,B 24.9187,C -2.0821,E1 24.9247,E2 -27.8176} C_DIS
LIN {X -50.6899,Y 89.3597,Z 102,A 115.3104,B 24.9213,C -2.0485,E1 24.9197,E2 -29.8842} C_DIS
LIN {X -53.9063,Y 87.4573,Z 102,A 117.3195,B 24.9218,C -2.0419,E1 24.9149,E2 -31.8839} C_DIS
LIN {X -56.487,Y 85.8109,Z 102,A 119.9108,B 24.9196,C -2.0708,E1 24.9087,E2 -34.5526} C_DIS
LIN {X -60.7859,Y 82.8213,Z 102,A 122.4342,B 24.9212,C -2.0503,E1 24.9031,E2 -37.0361} C_DIS
LIN {X -63.6762,Y 80.6203,Z 102,A 123.9919,B 24.9228,C -2.0291,E1 24.8998,E2 -38.5489} C_DIS
LIN {X -67.9469,Y 77.0568,Z 102,A 127.1685,B 24.9231,C -2.0248,E1 24.893,E2 -41.7275} C_DIS
LIN {X -70.6995,Y 74.539,Z 102,A 129.5541,B 24.9227,C -2.0308,E1 24.8881,E2 -44.1373} C_DIS
LIN {X -73.8187,Y 71.4502,Z 102,A 132.1087,B 24.9228,C -2.0287,E1 24.8831,E2 -46.6977} C_DIS
LIN {X -76.2469,Y 68.8542,Z 102,A 133.6394,B 24.9244,C -2.0076,E1 24.8803,E2 -48.1849} C_DIS
LIN {X -78.1095,Y 66.7324,Z 102,A 135.5448,B 24.9238,C -2.0153,E1 24.8768,E2 -50.1172} C_DIS
LIN {X -81.1478,Y 63.0037,Z 102,A 138.7139,B 24.9231,C -2.0255,E1 24.8713,E2 -53.3258} C_DIS
LIN {X -83.992,Y 59.1583,Z 102,A 140.3909,B 24.9263,C -1.983,E1 24.8687,E2 -54.9097} C_DIS
LIN {X -85.2719,Y 57.2983,Z 102,A 142.0289,B 24.9255,C -1.9929,E1 24.8661,E2 -56.5793} C_DIS
LIN {X -87.5611,Y 53.7359,Z 102,A 144.2096,B 24.9265,C -1.9798,E1 24.8629,E2 -58.7399} C_DIS
LIN {X -90.2468,Y 49.0899,Z 102,A 147.3516,B 24.9268,C -1.9764,E1 24.8586,E2 -61.8901} C_DIS
LIN {X -92.8786,Y 43.9117,Z 102,A 150.5364,B 24.9276,C -1.9647,E1 24.8546,E2 -65.0644} C_DIS
LIN {X -94.3337,Y 40.689,Z 102,A 152.5729,B 24.9279,C -1.961,E1 24.8523,E2 -67.1032} C_DIS
LIN {X -95.6952,Y 37.3733,Z 102,A 154.5302,B 24.9285,C -1.9535,E1 24.8503,E2 -69.0534} C_DIS
LIN {X -96.6208,Y 34.9115,Z 102,A 156.2497,B 24.9281,C -1.9578,E1 24.8486,E2 -70.793} C_DIS
LIN {X -98.112,Y 30.4685,Z 102,A 158.6625,B 24.9293,C -1.9426,E1 24.8466,E2 -73.1833} C_DIS
LIN {X -99.3239,Y 26.2555,Z 102,A 161.0064,B 24.9301,C -1.9313,E1 24.8448,E2 -75.5139} C_DIS
LIN {X -100.7584,Y 20.0602,Z 102,A 165.7449,B 24.9278,C -1.962,E1 24.842,E2 -80.3534} C_DIS
LIN {X -101.7369,Y 14.2804,Z 102,A 167.8299,B 24.9316,C -1.9097,E1 24.8412,E2 -82.3261} C_DIS
LIN {X -102.1153,Y 11.2638,Z 102,A 169.7564,B 24.9314,C -1.9123,E1 24.8406,E2 -84.2704} C_DIS
LIN {X -102.5042,Y 6.8684,Z 102,A 172.1009,B 24.9323,C -1.9003,E1 24.8401,E2 -86.6003} C_DIS
LIN {X -102.6739,Y 3.5368,Z 102,A 173.9966,B 24.9326,C -1.8955,E1 24.8398,E2 -88.496} C_DIS
LIN {X -102.7304,Y -0.9056,Z 102,A 176.7186,B 24.9326,C -1.896,E1 24.8398,E2 -91.2357} C_DIS
LIN {X -102.59,Y -5.4427,Z 102,A 178.9887,B 24.9338,C -1.8788,E1 24.8401,E2 -93.4783} C_DIS
LIN {X -102.3679,Y -8.68,Z 102,A -179.2821,B 24.9344,C -1.8701,E1 24.8404,E2 -95.1972} C_DIS
LIN {X -101.9235,Y -12.8839,Z 102,A -177.02,B 24.9352,C -1.8593,E1 24.8411,E2 -97.4471} C_DIS
LIN {X -101.4613,Y -16.1231,Z 102,A -174.6399,B 24.9342,C -1.873,E1 24.8421,E2 -99.8741} C_DIS
LIN {X -100.7481,Y -20.1102,Z 102,A -172.7406,B 24.9356,C -1.8533,E1 24.8431,E2 -101.7376} C_DIS
LIN {X -99.6585,Y -24.957,Z 102,A -169.7277,B 24.9356,C -1.8533,E1 24.845,E2 -104.7679} C_DIS
LIN {X -98.633,Y -28.7414,Z 102,A -167.604,B 24.9362,C -1.8444,E1 24.8466,E2 -106.8829} C_DIS
LIN {X -97.679,Y -31.8299,Z 102,A -165.7509,B 24.9365,C -1.8407,E1 24.8482,E2 -108.7379} C_DIS
LIN {X -96.4584,Y -35.3568,Z 102,A -163.6613,B 24.9369,C -1.8349,E1 24.8502,E2 -110.8254} C_DIS
LIN {X -94.8936,Y -39.3677,Z 102,A -160.5994,B 24.9357,C -1.8514,E1 24.8535,E2 -113.9438} C_DIS
LIN {X -93.1108,Y -43.4129,Z 102,A -158.7867,B 24.9378,C -1.8211,E1 24.8555,E2 -115.6941} C_DIS
LIN {X -91.8723,Y -45.9775,Z 102,A -156.9945,B 24.9376,C -1.8239,E1 24.8578,E2 -117.5028} C_DIS
LIN {X -89.7169,Y -50.0516,Z 102,A -154.688,B 24.9388,C -1.8075,E1 24.8608,E2 -119.7822} C_DIS
LIN {X -88.3139,Y -52.4881,Z 102,A -153.0008,B 24.9388,C -1.8075,E1 24.8632,E2 -121.4784} C_DIS
LIN {X -85.2565,Y -57.3212,Z 102,A -149.752,B 24.9392,C -1.8014,E1 24.8681,E2 -124.7289} C_DIS
LIN {X -83.0282,Y -60.5034,Z 102,A -147.6286,B 24.9396,C -1.7945,E1 24.8716,E2 -126.8461} C_DIS
LIN {X -80.6213,Y -63.6749,Z 102,A -145.4551,B 24.9401,C -1.7874,E1 24.8753,E2 -129.0131} C_DIS
LIN {X -78.3433,Y -66.458,Z 102,A -143.7236,B 24.9411,C -1.7728,E1 24.8783,E2 -130.7178} C_DIS
LIN {X -76.5429,Y -68.5235,Z 102,A -142.2318,B 24.9414,C -1.7681,E1 24.8811,E2 -132.205} C_DIS
LIN {X -74.2685,Y -70.9836,Z 102,A -139.9854,B 24.9408,C -1.7776,E1 24.8854,E2 -134.4839} C_DIS
LIN {X -71.9352,Y -73.3467,Z 102,A -138.1066,B 24.941,C -1.7746,E1 24.8891,E2 -136.3637} C_DIS
LIN {X -69.4394,Y -75.713,Z 102,A -136.237,B 24.9413,C -1.769,E1 24.8929,E2 -138.2274} C_DIS
LIN {X -64.1584,Y -80.2368,Z 102,A -132.2636,B 24.9416,C -1.765,E1 24.9014,E2 -142.2067} C_DIS
LIN {X -61.5432,Y -82.2604,Z 102,A -130.2799,B 24.9415,C -1.7669,E1 24.9059,E2 -144.202} C_DIS
LIN {X -58.1752,Y -84.6773,Z 102,A -128.1632,B 24.9422,C -1.7558,E1 24.9107,E2 -146.2995} C_DIS
LIN {X -55.1655,Y -86.6672,Z 102,A -126.2767,B 24.9427,C -1.748,E1 24.9151,E2 -148.1737} C_DIS
LIN {X -50.704,Y -89.3515,Z 102,A -123.122,B 24.9424,C -1.7531,E1 24.9227,E2 -151.35} C_DIS
LIN {X -47.3522,Y -91.1724,Z 102,A -121.229,B 24.9432,C -1.7416,E1 24.9273,E2 -153.2209} C_DIS
LIN {X -43.5879,Y -93.0293,Z 102,A -118.8397,B 24.9432,C -1.7406,E1 24.9333,E2 -155.614} C_DIS
LIN {X -40.2891,Y -94.5053,Z 102,A -116.9013,B 24.9436,C -1.7355,E1 24.9383,E2 -157.5449} C_DIS
LIN {X -33.2148,Y -97.2175,Z 102,A -112.6268,B 24.9436,C -1.7333,E1 24.9495,E2 -161.8231} C_DIS
LIN {X -28.7767,Y -98.6225,Z 102,A -109.8714,B 24.9434,C -1.7375,E1 24.9568,E2 -164.5931} C_DIS
LIN {X -25.0605,Y -99.632,Z 102,A -107.7333,B 24.9435,C -1.7358,E1 24.9626,E2 -166.7304} C_DIS
LIN {X -21.7165,Y -100.4127,Z 102,A -105.9305,B 24.9439,C -1.7306,E1 24.9675,E2 -168.5232} C_DIS
LIN {X -17.8779,Y -101.167,Z 102,A -103.7004,B 24.9439,C -1.7316,E1 24.9736,E2 -170.7581} C_DIS
LIN {X -14.3987,Y -101.72,Z 102,A -101.7216,B 24.9438,C -1.7316,E1 24.9791,E2 -172.7387} C_DIS
LIN {X -10.9046,Y -102.1539,Z 102,A -99.7963,B 24.9439,C -1.7299,E1 24.9844,E2 -174.6612} C_DIS
LIN {X -7.7684,Y -102.4408,Z 102,A -97.9352,B 24.9437,C -1.7339,E1 24.9896,E2 -176.5325} C_DIS
LIN {X -4.3587,Y -102.6416,Z 102,A -96.0428,B 24.9437,C -1.7336,E1 24.9949,E2 -178.4245} C_DIS
LIN {X -0.5517,Y -102.7326,Z 102,A -93.939,B 24.9437,C -1.7332,E1 25.0008,E2 -180.5276} C_DIS
LIN {X -0.5517,Y -102.7326,Z 102,A -93.939,B 24.9437,C -1.7332,E1 25.0008,E2 -180.5276} C_DIS
Enddeposition()
LIN {X 0.7138,Y -101.866,Z 102,A -93.9384,B 24.9445,C -1.7212,E1 25.0008,E2 -180.4998} C_DIS
Startdeposition()
$VEL.CP = VEL_PRINT
LIN {X -2.468,Y -101.8437,Z 102,A -96.0264,B 24.9452,C -1.7095,E1 24.9948,E2 -178.3838} C_DIS
LIN {X -6.3283,Y -101.6765,Z 102,A -98.1371,B 24.9451,C -1.7117,E1 24.9889,E2 -176.2779} C_DIS
LIN {X -9.8846,Y -101.3925,Z 102,A -100.229,B 24.9453,C -1.7086,E1 24.9831,E2 -174.1776} C_DIS
LIN {X -13.7722,Y -100.9382,Z 102,A -102.4745,B 24.9453,C -1.7073,E1 24.9768,E2 -171.9275} C_DIS
LIN {X -17.3261,Y -100.3891,Z 102,A -104.86,B 24.9462,C -1.6945,E1 24.9702,E2 -169.5092} C_DIS
LIN {X -21.0137,Y -99.6824,Z 102,A -106.2248,B 24.9444,C -1.7231,E1 24.9666,E2 -168.2108} C_DIS
LIN {X -24.8858,Y -98.7867,Z 102,A -108.9077,B 24.9454,C -1.7077,E1 24.9592,E2 -165.4875} C_DIS
LIN {X -30.2979,Y -97.2621,Z 102,A -111.5733,B 24.944,C -1.7282,E1 24.9522,E2 -162.8664} C_DIS
LIN {X -32.7119,Y -96.4771,Z 102,A -113.7543,B 24.9457,C -1.7017,E1 24.9463,E2 -160.6182} C_DIS
LIN {X -36.0355,Y -95.2854,Z 102,A -115.441,B 24.9449,C -1.7144,E1 24.9419,E2 -158.9583} C_DIS
LIN {X -39.9033,Y -93.7323,Z 102,A -117.7505,B 24.9447,C -1.7181,E1 24.936,E2 -156.6523} C_DIS
LIN {X -43.1151,Y -92.2983,Z 102,A -120.4741,B 24.9463,C -1.6934,E1 24.9289,E2 -153.8632} C_DIS
LIN {X -47.6583,Y -90.0367,Z 102,A -123.691,B 24.9468,C -1.6843,E1 24.9209,E2 -150.6157} C_DIS
LIN {X -53.2647,Y -86.8385,Z 102,A -126.1053,B 24.9437,C -1.7329,E1 24.9154,E2 -148.3097} C_DIS
LIN {X -56.7149,Y -84.6258,Z 102,A -128.229,B 24.9431,C -1.7431,E1 24.9105,E2 -146.2032} C_DIS
LIN {X -60.7121,Y -81.8062,Z 102,A -131.1875,B 24.9432,C -1.7403,E1 24.9037,E2 -143.2278} C_DIS
LIN {X -63.2908,Y -79.8259,Z 102,A -133.515,B 24.9442,C -1.7259,E1 24.8985,E2 -140.8575} C_DIS
LIN {X -66.0836,Y -77.5295,Z 102,A -135.0372,B 24.9427,C -1.7479,E1 24.8954,E2 -139.3817} C_DIS
LIN {X -68.6111,Y -75.3028,Z 102,A -136.9805,B 24.9427,C -1.7499,E1 24.8913,E2 -137.4355} C_DIS
LIN {X -71.1959,Y -72.8651,Z 102,A -139.0192,B 24.9424,C -1.7526,E1 24.8872,E2 -135.3948} C_DIS
LIN {X -73.6653,Y -70.3669,Z 102,A -141.4679,B 24.9432,C -1.7403,E1 24.8824,E2 -132.9062} C_DIS
LIN {X -76.1458,Y -67.6744,Z 102,A -142.9069,B 24.9415,C -1.7667,E1 24.8798,E2 -131.5235} C_DIS
LIN {X -77.9655,Y -65.5713,Z 102,A -144.5172,B 24.9414,C -1.7686,E1 24.8769,E2 -129.9105} C_DIS
LIN {X -79.7565,Y -63.3786,Z 102,A -146.1368,B 24.9412,C -1.7715,E1 24.874,E2 -128.2901} C_DIS
LIN {X -81.5245,Y -61.0872,Z 102,A -147.804,B 24.941,C -1.774,E1 24.8712,E2 -126.6212} C_DIS
LIN {X -83.7066,Y -58.061,Z 102,A -150.1588,B 24.9413,C -1.7704,E1 24.8674,E2 -124.246} C_DIS
LIN {X -86.5775,Y -53.6872,Z 102,A -153.1156,B 24.9408,C -1.7775,E1 24.8629,E2 -121.2913} C_DIS
LIN {X -88.6454,Y -50.202,Z 102,A -155.274,B 24.9401,C -1.7878,E1 24.8599,E2 -119.1461} C_DIS
LIN {X -90.3,Y -47.1583,Z 102,A -157.2149,B 24.9397,C -1.7934,E1 24.8574,E2 -117.2083} C_DIS
LIN {X -91.9027,Y -43.9522,Z 102,A -159.389,B 24.9397,C -1.7936,E1 24.8547,E2 -115.023} C_DIS
LIN {X -94.0583,Y -39.1297,Z 102,A -162.4755,B 24.9394,C -1.7982,E1 24.8513,E2 -111.9303} C_DIS
LIN {X -95.9512,Y -34.2275,Z 102,A -165.2348,B 24.9384,C -1.8136,E1 24.8486,E2 -109.1922} C_DIS
LIN {X -97.0824,Y -30.8732,Z 102,A -167.2289,B 24.938,C -1.8194,E1 24.8469,E2 -107.2006} C_DIS
LIN {X -98.1983,Y -27.1162,Z 102,A -169.4935,B 24.9376,C -1.8241,E1 24.8452,E2 -104.934} C_DIS
LIN {X -99.2076,Y -23.1469,Z 102,A -171.9084,B 24.9374,C -1.8274,E1 24.8436,E2 -102.5129} C_DIS
LIN {X -99.927,Y -19.819,Z 102,A -173.6916,B 24.9367,C -1.8378,E1 24.8426,E2 -100.7439} C_DIS
LIN {X -100.9856,Y -13.4123,Z 102,A -177.155,B 24.9354,C -1.8557,E1 24.8411,E2 -97.3028} C_DIS
LIN {X -101.5282,Y -8.3645,Z 102,A 179.8744,B 24.9351,C -1.8609,E1 24.8403,E2 -94.3266} C_DIS
LIN {X -101.7425,Y -5.1528,Z 102,A 177.477,B 24.9361,C -1.8468,E1 24.8399,E2 -91.8812} C_DIS
LIN {X -101.8627,Y -1.4315,Z 102,A 175.1973,B 24.9361,C -1.8473,E1 24.8398,E2 -89.589} C_DIS
LIN {X -101.8303,Y 2.918,Z 102,A 173.7674,B 24.9331,C -1.8896,E1 24.8398,E2 -88.2513} C_DIS
LIN {X -101.6872,Y 6.1358,Z 102,A 171.4617,B 24.9338,C -1.8786,E1 24.8402,E2 -85.9056} C_DIS
LIN {X -101.1699,Y 11.9389,Z 102,A 168.3972,B 24.9326,C -1.8964,E1 24.841,E2 -82.865} C_DIS
LIN {X -100.7145,Y 15.314,Z 102,A 165.553,B 24.9344,C -1.8713,E1 24.8422,E2 -79.9441} C_DIS
LIN {X -99.865,Y 20.1246,Z 102,A 163.8615,B 24.9312,C -1.9156,E1 24.8431,E2 -78.3484} C_DIS
Enddeposition()
END
